// TIA Portal project "Pierwszy_projekt" (V16)

(* hardware
DEVICE "S71500/ET200MP station_1"  S7-1500 station
   slot 0: "Rail_0"  Rack  6ES7 590-1***0-0AA0
   slot 1: "PLC_1"  CPU 1518F-4 PN/DP  6ES7 518-4FP00-3AB0  V2.8
      slot 3: "CPU display_1"  6ES7591-1BA00-0AA0
      slot 32768: "PROFINET interface_1"  X1
         slot 32769: "Port_1"  X1 P1
         slot 32770: "Port_2"  X1 P2
      slot 33024: "PROFINET interface_2"  X2
         slot 33025: "Port_1"  X2 P1
      slot 33280: "PROFINET interface GBIT_3"  X3
         slot 33281: "Port_1"  X3 P1
      slot 33536: "DP interface_1"  X4
      slot 34817: "Virtual CP interface port_1"  Virtual CP interface port  Virtual CP interface port
*)

// ===== PLC "PLC_1"  CPU 1518F-4 PN/DP =====

VAR_GLOBAL   // PLC tag table "Default tag table"
   "System_Byte" AT %MB1 : Byte;
   "FirstScan" AT %M1.0 : Bool;
   "DiagStatusUpdate" AT %M1.1 : Bool;
   "AlwaysTRUE" AT %M1.2 : Bool;
   "AlwaysFALSE" AT %M1.3 : Bool;
   "System_Byte(1)" AT %MB1 : Byte;
   "Clock_Byte" AT %MB0 : Byte;
   "Clock_10Hz" AT %M0.0 : Bool;
   "Clock_5Hz" AT %M0.1 : Bool;
   "Clock_2.5Hz" AT %M0.2 : Bool;
   "Clock_2Hz" AT %M0.3 : Bool;
   "Clock_1.25Hz" AT %M0.4 : Bool;
   "Clock_1Hz" AT %M0.5 : Bool;
   "Clock_0.625Hz" AT %M0.6 : Bool;
   "Clock_0.5Hz" AT %M0.7 : Bool;
   "11-PLC01-MANUAL" AT %Q1.6 : Bool;
   "11-PLC01-AUTOMAT" AT %Q1.7 : Bool;
   "11-PLC01-DISPLAY01" AT %QD58 : Real;
   "Tag_1" AT %M3.0 : Bool;
   "Tag_2" AT %M2.0 : Bool;
   "Tag_3" AT %M2.1 : Bool;
   "Tag_4" AT %M2.2 : Bool;
   "Tag_5" AT %M2.3 : Bool;
   "Tag_6" AT %QD43 : Real;
   "Tag_7" AT %QD44 : Real;
   "Tag_8" AT %M2.5 : Bool;
   "Tag_9" AT %M2.6 : Bool;
   "Tag_10" AT %M2.7 : Bool;
   "Tag_11" AT %M250.4 : Bool;
   "Tag_12" AT %M650.0 : Bool;
   "Tag_13" AT %M654.0 : Bool;
   "Tag_14" AT %M2.4 : Bool;
   "Tag_15" AT %M3.5 : Bool;
END_VAR

VAR_GLOBAL   // PLC tag table "Tag table from XML_1"
   "11-PLC01-CNR01-SQ01" AT %I0.0 : Bool;
   "11-PLC01-CNR01-SQ02" AT %I0.1 : Bool;
   "11-PLC01-CNR01-ENC-A" AT %I0.2 : Bool;
   "11-PLC01-CNR01-ENC-B" AT %I0.3 : Bool;
   "11-PLC01-CNR02-SQ01" AT %I0.4 : Bool;
   "11-PLC01-CNR02-SQ02" AT %I0.5 : Bool;
   "11-PLC01-CNR02-ENC-A" AT %I0.6 : Bool;
   "11-PLC01-CNR02-ENC-B" AT %I0.7 : Bool;
   "11-PLC01-CNR03-SQ01" AT %I1.0 : Bool;
   "11-PLC01-CNR03-SQ02" AT %I1.1 : Bool;
   "11-PLC01-CNR03-ENC-A" AT %I1.2 : Bool;
   "11-PLC01-CNR03-ENC-B" AT %I1.3 : Bool;
   "11-PLC01-B01(START)" AT %I3.5 : Bool;
   "11-PLC01-B02(STOP)" AT %I3.6 : Bool;
   "11-PLC01-B03(RESET)" AT %I3.7 : Bool;
   "11-PLC01-B04(MANUAL)" AT %I4.0 : Bool;
   "11-PLC01-B05(AUTOMAT)" AT %I4.1 : Bool;
   "FACTORY I/O (Running)" AT %I4.2 : Bool;
   "FACTORY I/O (Paused)" AT %I4.3 : Bool;
   "FACTORY I/O (Reset)" AT %Q1.5 : Bool;
   "11-PLC01-PX01(START)" AT %Q0.0 : Bool;
   "11-PLC01-PX02(STOP)" AT %Q0.1 : Bool;
   "11-PLC01-PX03(RESET)" AT %Q0.2 : Bool;
   "11-PLC01-CNR01-EM01" AT %Q0.3 : Bool;
   "11-PLC01-CNR03-RE01" AT %Q0.4 : Bool;
   "FACTORY I/O (Run)" AT %Q1.3 : Bool;
   "FACTORY I/O (Pause)" AT %Q1.4 : Bool;
   "FACTORY I/O (Time Scale)" AT %ID34 : Real;
   "11-PLC01-CNR01" AT %QD30 : Real;
   "11-PLC01-CNR02" AT %QD34 : Real;
   "11-PLC01-CNR03" AT %QD38 : Real;
   "FACTORY I/O (Camera Position)" AT %QD54 : DInt;
END_VAR

VAR_GLOBAL   // PLC tag table "Tag table from XML_2"
   "11-PLC01-TT01-SQ01" AT %I1.4 : Bool;
   "11-PLC01-TT01-SQ02" AT %I1.5 : Bool;
   "11-PLC01-TT01-SQ03" AT %I1.6 : Bool;
   "11-PLC01-TT01-SQ04" AT %I1.7 : Bool;
   "11-PLC01-TT01-SQ05" AT %I2.0 : Bool;
   "11-PLC01-CNR04-SQ01" AT %I2.1 : Bool;
   "11-PLC01-CNR04-SQ02" AT %I2.2 : Bool;
   "11-PLC01-CNR04-ENC-A" AT %I2.3 : Bool;
   "11-PLC01-CNR04-ENC-B" AT %I2.4 : Bool;
   "11-PLC01-CNR05-SQ01" AT %I2.5 : Bool;
   "11-PLC01-CNR05-SQ02" AT %I2.6 : Bool;
   "11-PLC01-CNR05-ENC-A" AT %I2.7 : Bool;
   "11-PLC01-CNR05-ENC-B" AT %I3.0 : Bool;
   "11-PLC01-CNR06-SQ01" AT %I3.1 : Bool;
   "11-PLC01-CNR06-SQ02" AT %I3.2 : Bool;
   "11-PLC01-CNR06-ENC-A" AT %I3.3 : Bool;
   "11-PLC01-CNR06-ENC-B" AT %I3.4 : Bool;
   "11-PLC01-CNR04-RE01" AT %Q0.5 : Bool;
   "11-PLC01-CNR05-RE01" AT %Q0.6 : Bool;
   "11-PLC01-CNR06-RE01" AT %Q0.7 : Bool;
   "11-PLC01-TT01-LEFT" AT %Q2.0 : Bool;
   "11-PLC01-TT01-RIGHT" AT %Q2.1 : Bool;
   "11-PLC01-TT01-FORWARD" AT %Q2.2 : Bool;
   "11-PLC01-TT01-BACKWARD" AT %Q2.3 : Bool;
   "11-PLC01-CNR03-FLC01" AT %ID30 : Real;
   "11-PLC01-CNR04" AT %QD42 : Real;
   "11-PLC01-CNR05" AT %QD46 : Real;
   "11-PLC01-CNR06" AT %QD50 : Real;
END_VAR

DATA_BLOCK "Main_Safety_RTG1_DB"   // DB1, F_DB
{ S7_Optimized_Access := 'TRUE' }
NAME : FUSI
VERSION : 0.1
// stored: InstanceOfName Main_Safety_RTG1
"Main_Safety_RTG1"
BEGIN
END_DATA_BLOCK

DATA_BLOCK "FB_Conveyor_DB"   // DB2
{ S7_Optimized_Access := 'TRUE' }
VERSION : 0.1
// stored: InstanceOfName FB_Conveyor
"FB_Conveyor"
BEGIN
END_DATA_BLOCK

DATA_BLOCK "FB_Conveyor_DB_2"   // DB3
{ S7_Optimized_Access := 'TRUE' }
VERSION : 0.1
// stored: InstanceOfName FB_Conveyor
"FB_Conveyor"
BEGIN
END_DATA_BLOCK

DATA_BLOCK "DB_Manual"   // DB6
{ S7_Optimized_Access := 'TRUE' }
VERSION : 0.1
   VAR
      "11-CNR01-CONV" : Struct
         SelectManualMode : Bool := TRUE;
         StartStop : Bool := TRUE;
         SetSpeed : Int := 80;
      END_STRUCT;
      "11-CNR02-CONV" : Struct
         SelectManual : Bool := TRUE;
         StartStop : Bool := TRUE;
         SetSpeed : Int := 80;
      END_STRUCT;
      "11-CNRO3-CONV" : Struct
         SelectManualMode : Bool := TRUE;
         StartStop : Bool := TRUE;
         SetSpeed : Int := 100;
      END_STRUCT;
   END_VAR
BEGIN
END_DATA_BLOCK

DATA_BLOCK "FB_Inverter_DB"   // DB7
{ S7_Optimized_Access := 'TRUE' }
VERSION : 0.1
// stored: InstanceOfName FB_Inverter
"FB_Inverter"
BEGIN
END_DATA_BLOCK

DATA_BLOCK "FB_Conveyor_DB_1"   // DB8
{ S7_Optimized_Access := 'TRUE' }
VERSION : 0.1
// stored: InstanceOfName FB_Conveyor
"FB_Conveyor"
BEGIN
END_DATA_BLOCK

DATA_BLOCK "DB_Signals"   // DB9
{ S7_Optimized_Access := 'TRUE' }
VERSION : 0.1
   VAR
      "11-CNR01-VFD" : Struct
         RunForward : Bool;
         RunRevers : Bool;
         ConveyorSpeedSetPoint : Real;
      END_STRUCT;
      "11-CNR02-VFD" : Struct
         RunForward : Bool;
         RunRevers : Bool;
         ConveyorSpeedSetPoint : Real;
      END_STRUCT;
      "11-CNR03-VFD" : Struct
         RunForward : Bool;
         RunRevrs : Bool;
         ConveyorSpeedSetPoint : Real;
      END_STRUCT;
   END_VAR
BEGIN
END_DATA_BLOCK

DATA_BLOCK "DB_Configuration"   // DB10
{ S7_Optimized_Access := 'TRUE' }
VERSION : 0.1
   VAR
      "11-CNR01-VFD" : Struct
         InterlockForwad : Bool := TRUE;
         InterockReverse : Bool;
      END_STRUCT;
      "11-CNR02-VDF" : Struct
         InterlockForwad : Bool := TRUE;
         InterockReverse : Bool;
      END_STRUCT;
      "11-CNR03-VDF" : Struct
         InterlockForwad : Bool := TRUE;
         InterockReverse : Bool;
      END_STRUCT;
   END_VAR
BEGIN
END_DATA_BLOCK

DATA_BLOCK "FB_Inverter_DB_1"   // DB11
{ S7_Optimized_Access := 'TRUE' }
VERSION : 0.1
// stored: InstanceOfName FB_Inverter
"FB_Inverter"
BEGIN
END_DATA_BLOCK

DATA_BLOCK "FB_Inverter_DB_2"   // DB12
{ S7_Optimized_Access := 'TRUE' }
VERSION : 0.1
// stored: InstanceOfName FB_Inverter
"FB_Inverter"
BEGIN
END_DATA_BLOCK

DATA_BLOCK "FB_TurnTable_DB"   // DB13
{ S7_Optimized_Access := 'TRUE' }
VERSION : 0.1
// stored: InstanceOfName FB_TurnTable
"FB_TurnTable"
BEGIN
END_DATA_BLOCK

DATA_BLOCK "FB_Control_DB"   // DB14
{ S7_Optimized_Access := 'TRUE' }
VERSION : 0.1
// stored: InstanceOfName FB_Control
"FB_Control"
BEGIN
END_DATA_BLOCK

DATA_BLOCK "FB_Control_DB_1"   // DB15
{ S7_Optimized_Access := 'TRUE' }
VERSION : 0.1
// stored: InstanceOfName FB_Control
"FB_Control"
BEGIN
END_DATA_BLOCK

DATA_BLOCK "DB_Control"   // DB16
{ S7_Optimized_Access := 'TRUE' }
VERSION : 0.1
   VAR
      StartCommand : Bool := false;
      StopCommand : Bool;
      StartFeedback : Bool := false;
      StopFeedback : Bool;
      ManualFeedback : Bool;
   END_VAR
BEGIN
END_DATA_BLOCK

DATA_BLOCK "IDB_FIFO"   // DB20
{ S7_Optimized_Access := 'TRUE' }
VERSION : 0.1
   VAR
      Static_1 : Array[0..10] of Real;
      Arrey_return : Int;
      Array_Dest : Array[0..10] of Real;
      Array_Input : Array[0..5] of Real;
      Array_endofqueue : Array[0..10] of Real;
   END_VAR
BEGIN
END_DATA_BLOCK

DATA_BLOCK "FD_FIFO_DB"   // DB22
{ S7_Optimized_Access := 'TRUE' }
VERSION : 0.1
// stored: InstanceOfName FD_FIFO
"FD_FIFO"
BEGIN
END_DATA_BLOCK

DATA_BLOCK "FB_Chute_DB- smallpackage"   // DB25
{ S7_Optimized_Access := 'TRUE' }
VERSION : 0.1
// stored: InstanceOfName FB_Chute
"FB_Chute"
BEGIN
END_DATA_BLOCK

DATA_BLOCK "FB_Chute_DB-mediumpackage"   // DB26
{ S7_Optimized_Access := 'TRUE' }
VERSION : 0.1
// stored: InstanceOfName FB_Chute
"FB_Chute"
BEGIN
END_DATA_BLOCK

DATA_BLOCK "FB_Chute_DB-bigpackage"   // DB27
{ S7_Optimized_Access := 'TRUE' }
VERSION : 0.1
// stored: InstanceOfName FB_Chute
"FB_Chute"
BEGIN
END_DATA_BLOCK

DATA_BLOCK "DB_Chute"   // DB30
{ S7_Optimized_Access := 'TRUE' }
VERSION : 0.1
   VAR
      "Small Package" : Int;
      "Medium Package" : Int;
      "Big Package" : Int;
   END_VAR
BEGIN
END_DATA_BLOCK

// folder: System blocks/Program resources

DATA_BLOCK "StartButtonCount_DB"   // DB4
{ S7_Optimized_Access := 'TRUE' }
AUTHOR : Simatic
FAMILY : IEC
NAME : CNTR
VERSION : 1.0
// stored: InstanceOfName IEC_COUNTER
"IEC_COUNTER"
BEGIN
END_DATA_BLOCK

DATA_BLOCK "DelayStartDB"   // DB5
{ S7_Optimized_Access := 'TRUE' }
AUTHOR : Simatic
FAMILY : IEC
NAME : IEC_TMR
VERSION : 1.0
// stored: InstanceOfName IEC_TIMER
"IEC_TIMER"
BEGIN
END_DATA_BLOCK

DATA_BLOCK "IEC_Counter_0_DB"   // DB17
{ S7_Optimized_Access := 'TRUE' }
AUTHOR : Simatic
FAMILY : IEC
NAME : CNTR
VERSION : 1.0
// stored: InstanceOfName IEC_COUNTER
"IEC_COUNTER"
BEGIN
END_DATA_BLOCK

DATA_BLOCK "IEC_Counter_0_DB_1"   // DB18
{ S7_Optimized_Access := 'TRUE' }
AUTHOR : Simatic
FAMILY : IEC
NAME : CNTR
VERSION : 1.0
// stored: InstanceOfName IEC_COUNTER
"IEC_COUNTER"
BEGIN
END_DATA_BLOCK

DATA_BLOCK "IEC_Counter_0_DB_2"   // DB19
{ S7_Optimized_Access := 'TRUE' }
AUTHOR : Simatic
FAMILY : IEC
NAME : CNTR
VERSION : 1.0
// stored: InstanceOfName IEC_COUNTER
"IEC_COUNTER"
BEGIN
END_DATA_BLOCK

DATA_BLOCK "IEC_Counter_0_DB_3"   // DB21
{ S7_Optimized_Access := 'TRUE' }
AUTHOR : Simatic
FAMILY : IEC
NAME : CNTR
VERSION : 1.0
// stored: InstanceOfName IEC_COUNTER
"IEC_COUNTER"
BEGIN
END_DATA_BLOCK

DATA_BLOCK "IEC_Counter_0_DB_4"   // DB24
{ S7_Optimized_Access := 'TRUE' }
AUTHOR : Simatic
FAMILY : IEC
NAME : CNTR
VERSION : 1.0
// stored: InstanceOfName IEC_COUNTER
"IEC_COUNTER"
BEGIN
END_DATA_BLOCK

DATA_BLOCK "IEC_Counter_0_DB_5"   // DB28
{ S7_Optimized_Access := 'TRUE' }
AUTHOR : Simatic
FAMILY : IEC
NAME : CNTR
VERSION : 1.0
// stored: InstanceOfName IEC_COUNTER
"IEC_COUNTER"
BEGIN
END_DATA_BLOCK

DATA_BLOCK "IEC_Counter_0_DB_6"   // DB29
{ S7_Optimized_Access := 'TRUE' }
AUTHOR : Simatic
FAMILY : IEC
NAME : CNTR
VERSION : 1.0
// stored: InstanceOfName IEC_COUNTER
"IEC_COUNTER"
BEGIN
END_DATA_BLOCK

// folder: (top level)

FUNCTION_BLOCK "Main_Safety_RTG1"   // FB1, F_FBD
{ S7_Optimized_Access := 'TRUE' }
BEGIN
END_FUNCTION_BLOCK

FUNCTION_BLOCK "FB_Conveyor"   // FB2, LAD
{ S7_Optimized_Access := 'TRUE' }
VERSION : 0.1
   VAR_INPUT
      ir_ConveyorSpeed : Real;
      ix_PEC_BOS : Bool;
      ix_PEC_EOS : Bool;
   END_VAR
   VAR_OUTPUT
      qx_FlowStop : Bool;
   END_VAR
   VAR_IN_OUT
      iqx_StartStop : Bool;
      iqi_SetSpeed : Int;
      iqx_SelectManualMode : Bool;
      iqr_InverterSpeedSetpoint : Real;
      iqx_InverterRunForward : Bool;
      iqx_InverterRunReverse : Bool;
      iqx_ControlStart : Bool;
      iqx_ControlStop : Bool;
      iqx_ControlManual : Bool;
   END_VAR
   VAR
      sx_manual : Bool;
      sx_Automatic : Bool;
      sx_FlowStop : Bool;
   END_VAR
   VAR_TEMP
      tr_SpeedPoint : Real;
      tr_SpeedProcent : Int;
   END_VAR
   VAR_TEMP   // added for the SCL form of the ladder/FBD networks
      _w1 : Bool;
      _w2 : Bool;
      _w3 : Bool;
   END_VAR
BEGIN

REGION Network 1
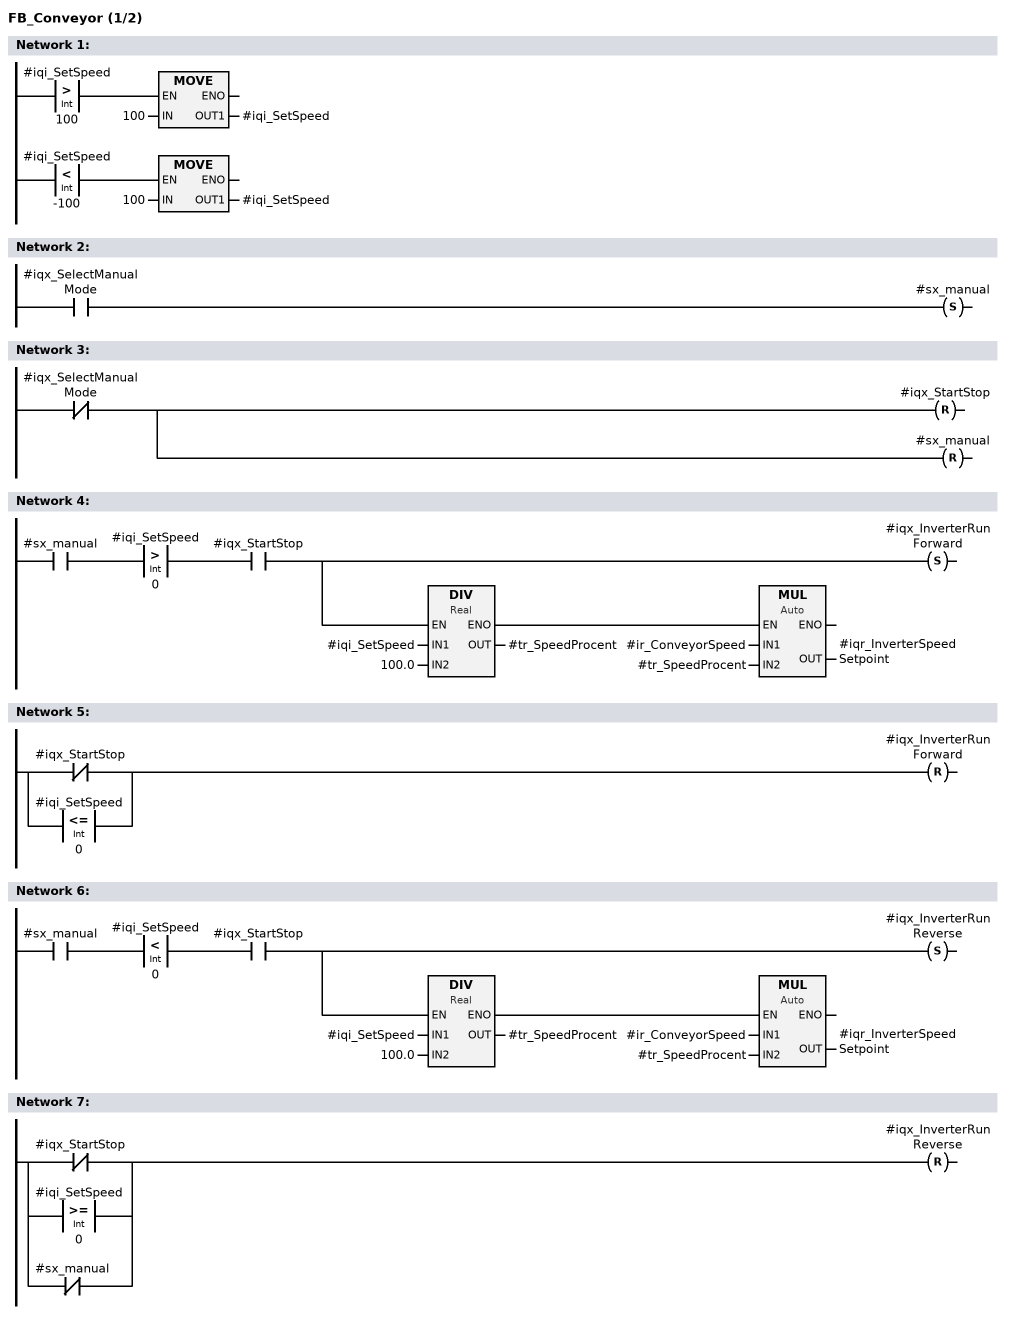
   RUNG wire#powerrail
      { S7_Templates := "SrcType := Int" } GT_Contact(in1 := #iqi_SetSpeed, in2 := 100)
      Move(in := 100, out1 => #iqi_SetSpeed)
   END_RUNG
   RUNG wire#powerrail
      { S7_Templates := "SrcType := Int" } LT_Contact(in1 := #iqi_SetSpeed, in2 := -100)
      Move(in := 100, out1 => #iqi_SetSpeed)
   END_RUNG
   // the same network as SCL:
   IF #iqi_SetSpeed > 100 THEN #iqi_SetSpeed := 100; END_IF;
   IF #iqi_SetSpeed < (-100) THEN #iqi_SetSpeed := 100; END_IF;
END_REGION

REGION Network 2
   RUNG wire#powerrail
      Contact( #iqx_SelectManualMode )
      S_Coil( #sx_manual )
   END_RUNG
   // the same network as SCL:
   IF #iqx_SelectManualMode THEN #sx_manual := TRUE; END_IF;
END_REGION

REGION Network 3
   RUNG wire#powerrail
      I_Contact( #iqx_SelectManualMode )
      wire#w1
      R_Coil( #iqx_StartStop )
   END_RUNG
   RUNG wire#w1
      R_Coil( #sx_manual )
   END_RUNG
   // the same network as SCL:
   IF NOT #iqx_SelectManualMode THEN
       #iqx_StartStop := FALSE;
       #sx_manual := FALSE;
   END_IF;
END_REGION

REGION Network 4
   RUNG wire#powerrail
      Contact( #sx_manual )
      { S7_Templates := "SrcType := Int" } GT_Contact(in1 := #iqi_SetSpeed, in2 := 0)
      Contact( #iqx_StartStop )
      wire#w1
      S_Coil( #iqx_InverterRunForward )
   END_RUNG
   RUNG wire#w1
      { S7_Templates := "SrcType := Real" } Div(in1 := #iqi_SetSpeed, in2 := 100.0, out => #tr_SpeedProcent)
      Mul(in1 := #ir_ConveyorSpeed, in2 := #tr_SpeedProcent, out => #iqr_InverterSpeedSetpoint)
   END_RUNG
   // the same network as SCL:
   IF #sx_manual AND (#iqi_SetSpeed > 0) AND #iqx_StartStop THEN
       #iqx_InverterRunForward := TRUE;
       #tr_SpeedProcent := #iqi_SetSpeed / 100.0;
       #iqr_InverterSpeedSetpoint := #ir_ConveyorSpeed * #tr_SpeedProcent;
   END_IF;
END_REGION

REGION Network 5
   RUNG wire#powerrail
      I_Contact( #iqx_StartStop )
      wire#w1
      R_Coil( #iqx_InverterRunForward )
   END_RUNG
   RUNG wire#powerrail
      { S7_Templates := "SrcType := Int" } LE_Contact(in1 := #iqi_SetSpeed, in2 := 0)
   END_RUNG wire#w1
   // the same network as SCL:
   IF NOT #iqx_StartStop OR (#iqi_SetSpeed <= 0) THEN #iqx_InverterRunForward := FALSE; END_IF;
END_REGION

REGION Network 6
   RUNG wire#powerrail
      Contact( #sx_manual )
      { S7_Templates := "SrcType := Int" } LT_Contact(in1 := #iqi_SetSpeed, in2 := 0)
      Contact( #iqx_StartStop )
      wire#w1
      S_Coil( #iqx_InverterRunReverse )
   END_RUNG
   RUNG wire#w1
      { S7_Templates := "SrcType := Real" } Div(in1 := #iqi_SetSpeed, in2 := 100.0, out => #tr_SpeedProcent)
      Mul(in1 := #ir_ConveyorSpeed, in2 := #tr_SpeedProcent, out => #iqr_InverterSpeedSetpoint)
   END_RUNG
   // the same network as SCL:
   IF #sx_manual AND (#iqi_SetSpeed < 0) AND #iqx_StartStop THEN
       #iqx_InverterRunReverse := TRUE;
       #tr_SpeedProcent := #iqi_SetSpeed / 100.0;
       #iqr_InverterSpeedSetpoint := #ir_ConveyorSpeed * #tr_SpeedProcent;
   END_IF;
END_REGION

REGION Network 7
   RUNG wire#powerrail
      I_Contact( #iqx_StartStop )
      wire#w1
      R_Coil( #iqx_InverterRunReverse )
   END_RUNG
   RUNG wire#powerrail
      { S7_Templates := "SrcType := Int" } GE_Contact(in1 := #iqi_SetSpeed, in2 := 0)
   END_RUNG wire#w1
   RUNG wire#powerrail
      I_Contact( #sx_manual )
   END_RUNG wire#w1
   // the same network as SCL:
   IF NOT #iqx_StartStop OR (#iqi_SetSpeed >= 0) OR NOT #sx_manual THEN
       #iqx_InverterRunReverse := FALSE;
   END_IF;
END_REGION

REGION Network 8
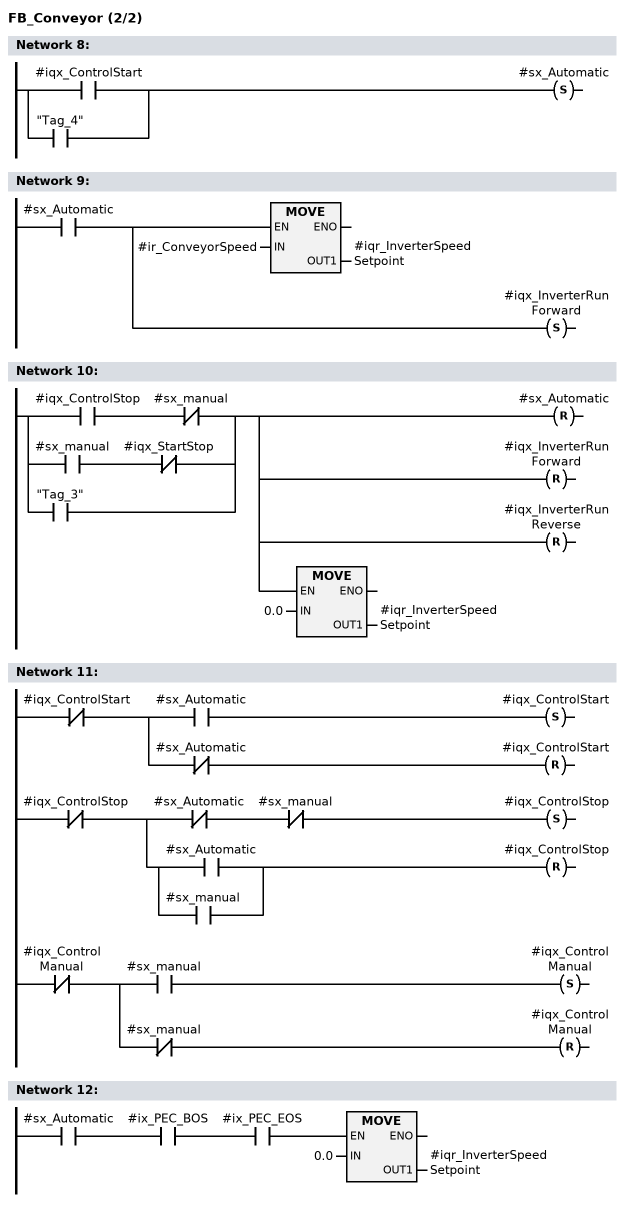
   RUNG wire#powerrail
      Contact( #iqx_ControlStart )
      wire#w1
      S_Coil( #sx_Automatic )
   END_RUNG
   RUNG wire#powerrail
      Contact( "Tag_4" )
   END_RUNG wire#w1
   // the same network as SCL:
   IF #iqx_ControlStart OR "Tag_4" THEN #sx_Automatic := TRUE; END_IF;
END_REGION

REGION Network 9
   RUNG wire#powerrail
      Contact( #sx_Automatic )
      wire#w1
      Move(in := #ir_ConveyorSpeed, out1 => #iqr_InverterSpeedSetpoint)
   END_RUNG
   RUNG wire#w1
      S_Coil( #iqx_InverterRunForward )
   END_RUNG
   // the same network as SCL:
   IF #sx_Automatic THEN
       #iqr_InverterSpeedSetpoint := #ir_ConveyorSpeed;
       #iqx_InverterRunForward := TRUE;
   END_IF;
END_REGION

REGION Network 10
   RUNG wire#powerrail
      Contact( #iqx_ControlStop )
      I_Contact( #sx_manual )
      wire#w1
      R_Coil( #sx_Automatic )
   END_RUNG
   RUNG wire#powerrail
      Contact( #sx_manual )
      I_Contact( #iqx_StartStop )
   END_RUNG wire#w1
   RUNG wire#powerrail
      Contact( "Tag_3" )
   END_RUNG wire#w1
   RUNG wire#w1
      R_Coil( #iqx_InverterRunForward )
   END_RUNG
   RUNG wire#w1
      R_Coil( #iqx_InverterRunReverse )
   END_RUNG
   RUNG wire#w1
      Move(in := 0.0, out1 => #iqr_InverterSpeedSetpoint)
   END_RUNG
   // the same network as SCL:
   IF (#iqx_ControlStop AND NOT #sx_manual) OR (#sx_manual AND NOT #iqx_StartStop) OR "Tag_3" THEN
       #sx_Automatic := FALSE;
       #iqx_InverterRunForward := FALSE;
       #iqx_InverterRunReverse := FALSE;
       #iqr_InverterSpeedSetpoint := 0.0;
   END_IF;
END_REGION

REGION Network 11
   RUNG wire#powerrail
      I_Contact( #iqx_ControlStart )
      wire#w1
      Contact( #sx_Automatic )
      S_Coil( #iqx_ControlStart )
   END_RUNG
   RUNG wire#w1
      I_Contact( #sx_Automatic )
      R_Coil( #iqx_ControlStart )
   END_RUNG
   RUNG wire#powerrail
      I_Contact( #iqx_ControlStop )
      wire#w2
      I_Contact( #sx_Automatic )
      I_Contact( #sx_manual )
      S_Coil( #iqx_ControlStop )
   END_RUNG
   RUNG wire#w2
      Contact( #sx_Automatic )
      wire#w3
      R_Coil( #iqx_ControlStop )
   END_RUNG
   RUNG wire#w2
      Contact( #sx_manual )
   END_RUNG wire#w3
   RUNG wire#powerrail
      I_Contact( #iqx_ControlManual )
      wire#w4
      Contact( #sx_manual )
      S_Coil( #iqx_ControlManual )
   END_RUNG
   RUNG wire#w4
      I_Contact( #sx_manual )
      R_Coil( #iqx_ControlManual )
   END_RUNG
   // the same network as SCL:
   #_w1 := NOT #iqx_ControlStart;
   IF NOT #iqx_ControlStart AND #sx_Automatic THEN #iqx_ControlStart := TRUE; END_IF;
   IF #_w1 AND NOT #sx_Automatic THEN #iqx_ControlStart := FALSE; END_IF;
   #_w2 := NOT #iqx_ControlStop;
   IF NOT #iqx_ControlStop AND NOT #sx_Automatic AND NOT #sx_manual THEN #iqx_ControlStop := TRUE; END_IF;
   IF #_w2 AND (#sx_Automatic OR #sx_manual) THEN #iqx_ControlStop := FALSE; END_IF;
   #_w3 := NOT #iqx_ControlManual;
   IF NOT #iqx_ControlManual AND #sx_manual THEN #iqx_ControlManual := TRUE; END_IF;
   IF #_w3 AND NOT #sx_manual THEN #iqx_ControlManual := FALSE; END_IF;
END_REGION

REGION Network 12
   RUNG wire#powerrail
      Contact( #sx_Automatic )
      Contact( #ix_PEC_BOS )
      Contact( #ix_PEC_EOS )
      Move(in := 0.0, out1 => #iqr_InverterSpeedSetpoint)
   END_RUNG
   // the same network as SCL:
   IF #sx_Automatic AND #ix_PEC_BOS AND #ix_PEC_EOS THEN #iqr_InverterSpeedSetpoint := 0.0; END_IF;
END_REGION
END_FUNCTION_BLOCK

FUNCTION_BLOCK "FB_Inverter"   // FB3, LAD
{ S7_Optimized_Access := 'TRUE' }
VERSION : 0.1
   VAR_INPUT
      ix_InterlockForward : Bool;
      Ix_InterlockReverse : Bool;
      Ir_ConveyorSpeedSetpoint : Real;
   END_VAR
   VAR_OUTPUT
      qr_InverterSpeed : Real;
   END_VAR
   VAR_IN_OUT
      iqx_InverterRunForward : Bool;
      iqx_InverterRunReverse : Bool;
   END_VAR
   VAR
      sx_RunForward : Bool;
      sx_RunReverse : Bool;
   END_VAR
BEGIN

REGION Network 1
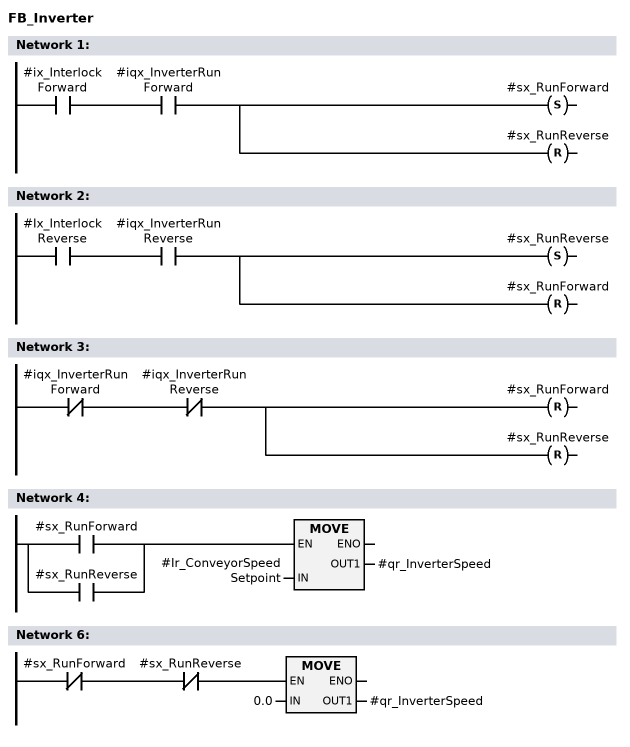
   RUNG wire#powerrail
      Contact( #ix_InterlockForward )
      Contact( #iqx_InverterRunForward )
      wire#w1
      S_Coil( #sx_RunForward )
   END_RUNG
   RUNG wire#w1
      R_Coil( #sx_RunReverse )
   END_RUNG
   // the same network as SCL:
   IF #ix_InterlockForward AND #iqx_InverterRunForward THEN
       #sx_RunForward := TRUE;
       #sx_RunReverse := FALSE;
   END_IF;
END_REGION

REGION Network 2
   RUNG wire#powerrail
      Contact( #Ix_InterlockReverse )
      Contact( #iqx_InverterRunReverse )
      wire#w1
      S_Coil( #sx_RunReverse )
   END_RUNG
   RUNG wire#w1
      R_Coil( #sx_RunForward )
   END_RUNG
   // the same network as SCL:
   IF #Ix_InterlockReverse AND #iqx_InverterRunReverse THEN
       #sx_RunReverse := TRUE;
       #sx_RunForward := FALSE;
   END_IF;
END_REGION

REGION Network 3
   RUNG wire#powerrail
      I_Contact( #iqx_InverterRunForward )
      I_Contact( #iqx_InverterRunReverse )
      wire#w1
      R_Coil( #sx_RunForward )
   END_RUNG
   RUNG wire#w1
      R_Coil( #sx_RunReverse )
   END_RUNG
   // the same network as SCL:
   IF NOT #iqx_InverterRunForward AND NOT #iqx_InverterRunReverse THEN
       #sx_RunForward := FALSE;
       #sx_RunReverse := FALSE;
   END_IF;
END_REGION

REGION Network 4
   RUNG wire#powerrail
      Contact( #sx_RunForward )
      wire#w1
      Move(in := #Ir_ConveyorSpeedSetpoint, out1 => #qr_InverterSpeed)
   END_RUNG
   RUNG wire#powerrail
      Contact( #sx_RunReverse )
   END_RUNG wire#w1
   // the same network as SCL:
   IF #sx_RunForward OR #sx_RunReverse THEN #qr_InverterSpeed := #Ir_ConveyorSpeedSetpoint; END_IF;
END_REGION

REGION Network 6
   RUNG wire#powerrail
      I_Contact( #sx_RunForward )
      I_Contact( #sx_RunReverse )
      Move(in := 0.0, out1 => #qr_InverterSpeed)
   END_RUNG
   // the same network as SCL:
   IF NOT #sx_RunForward AND NOT #sx_RunReverse THEN #qr_InverterSpeed := 0.0; END_IF;
END_REGION
END_FUNCTION_BLOCK

FUNCTION_BLOCK "FB_Control"   // FB4, LAD
{ S7_Optimized_Access := 'TRUE' }
VERSION : 0.1
   VAR_IN_OUT
      iqx_StartHMICommand : Bool;
      iqx_StopHMICommand : Bool;
      iqx_StartFeedback : Bool;
      iqx_StopFeedback : Bool;
      iqx_ManualFeedback : Bool;
   END_VAR
   VAR
      sudi_SignalingTime : Time := T#300ms;
      sx_StartRequest : Bool;
      s_TON_Timer : TON_TIME;
   END_VAR
BEGIN

REGION Network 1
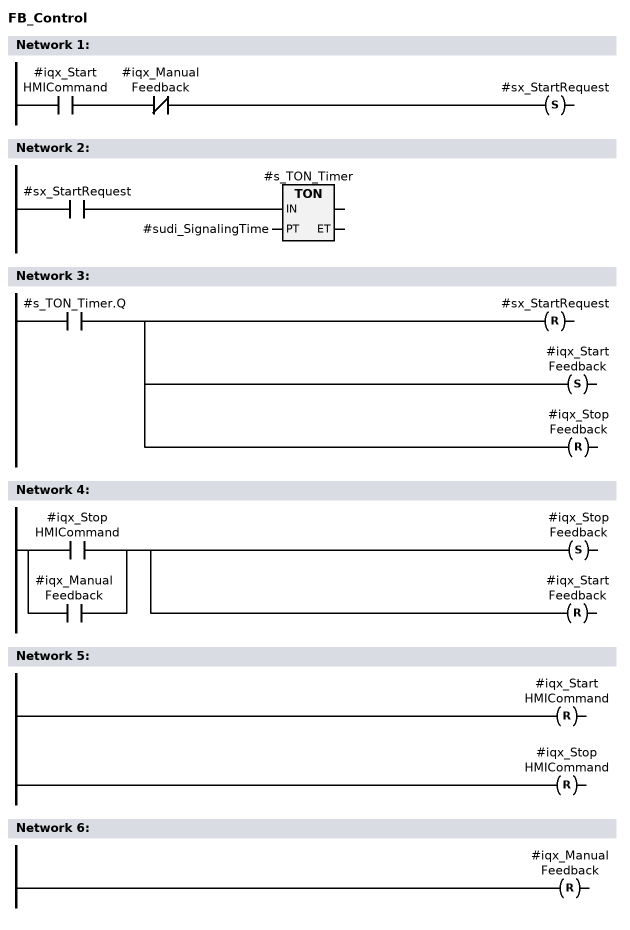
   RUNG wire#powerrail
      Contact( #iqx_StartHMICommand )
      I_Contact( #iqx_ManualFeedback )
      S_Coil( #sx_StartRequest )
   END_RUNG
   // the same network as SCL:
   IF #iqx_StartHMICommand AND NOT #iqx_ManualFeedback THEN #sx_StartRequest := TRUE; END_IF;
END_REGION

REGION Network 2
   #s_TON_Timer(IN := #sx_StartRequest, PT := #sudi_SignalingTime);   // TON
END_REGION

REGION Network 3
   RUNG wire#powerrail
      Contact( #s_TON_Timer.Q )
      wire#w1
      R_Coil( #sx_StartRequest )
   END_RUNG
   RUNG wire#w1
      S_Coil( #iqx_StartFeedback )
   END_RUNG
   RUNG wire#w1
      R_Coil( #iqx_StopFeedback )
   END_RUNG
   // the same network as SCL:
   IF #s_TON_Timer.Q THEN
       #sx_StartRequest := FALSE;
       #iqx_StartFeedback := TRUE;
       #iqx_StopFeedback := FALSE;
   END_IF;
END_REGION

REGION Network 4
   RUNG wire#powerrail
      Contact( #iqx_StopHMICommand )
      wire#w1
      S_Coil( #iqx_StopFeedback )
   END_RUNG
   RUNG wire#powerrail
      Contact( #iqx_ManualFeedback )
   END_RUNG wire#w1
   RUNG wire#w1
      R_Coil( #iqx_StartFeedback )
   END_RUNG
   // the same network as SCL:
   IF #iqx_StopHMICommand OR #iqx_ManualFeedback THEN
       #iqx_StopFeedback := TRUE;
       #iqx_StartFeedback := FALSE;
   END_IF;
END_REGION

REGION Network 5
   RUNG wire#powerrail
      R_Coil( #iqx_StartHMICommand )
   END_RUNG
   RUNG wire#powerrail
      R_Coil( #iqx_StopHMICommand )
   END_RUNG
   // the same network as SCL:
   #iqx_StartHMICommand := FALSE;
   #iqx_StopHMICommand := FALSE;
END_REGION

REGION Network 6
   RUNG wire#powerrail
      R_Coil( #iqx_ManualFeedback )
   END_RUNG
   // the same network as SCL:
   #iqx_ManualFeedback := FALSE;
END_REGION
END_FUNCTION_BLOCK

FUNCTION_BLOCK "FB_TurnTable"   // FB5, LAD
{ S7_Optimized_Access := 'TRUE' }
VERSION : 0.1
   VAR_INPUT
      ix_PEC_BigPackage_1 : Bool;
      ix_PEC_BigPackage_2 : Bool;
      ix_PEC_MediumPackage_1 : Bool;
      ix_PEC_MediumPackage_2 : Bool;
      ix_PEC_SmallPackage_1 : Bool;
      ix_PEC_SmallPackage_2 : Bool;
      ix_PEC_DetectPackage_1 : Bool;
      ix_PEC_DetectPackage_2 : Bool;
      ix_PEC_90Degree : Bool;
      ix_PEC_DiagonallyTT : Bool;
      ix_Reset : Bool;
   END_VAR
   VAR_OUTPUT
      qx_TTForward : Bool;
      qx_TTBackward : Bool;
      qx_TTLeft : Bool;
      qx_TTRight : Bool;
   END_VAR
   VAR_IN_OUT
      sx_Automatic_2 : Bool;
   END_VAR
   VAR
      sx_Automatic : Bool;
   END_VAR
   VAR_TEMP   // added for the SCL form of the ladder/FBD networks
      _w1 : Bool;
   END_VAR
BEGIN

REGION Network 1
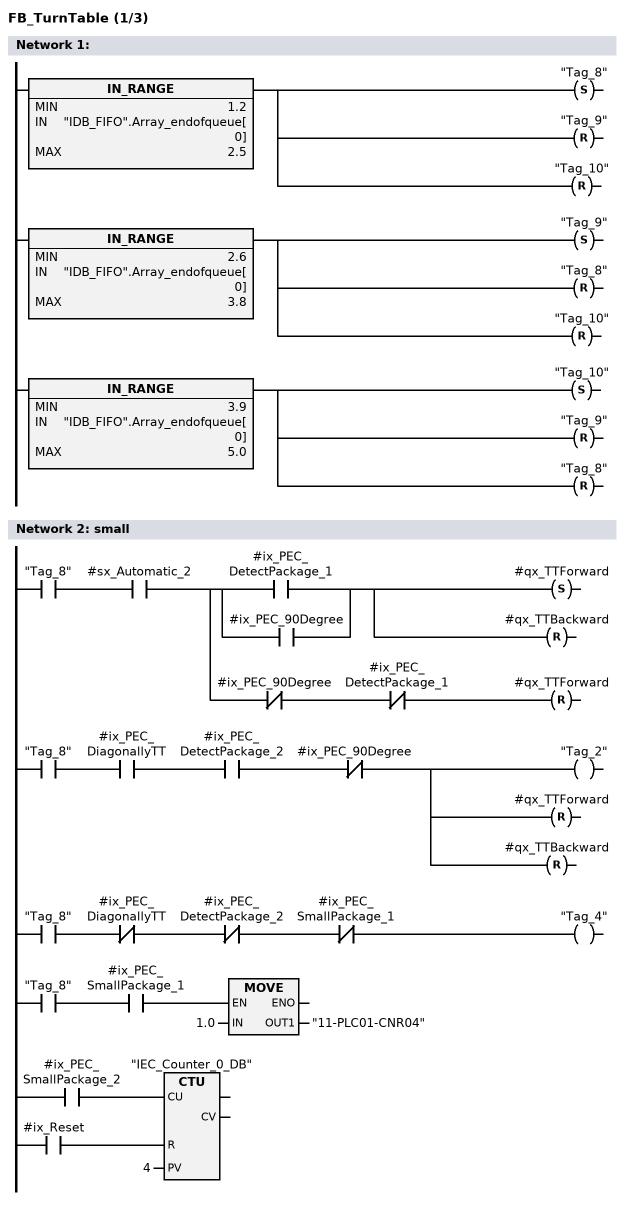
   RUNG wire#powerrail
      { S7_Templates := "SrcType := Real" } InRange(min := 1.2, in := "IDB_FIFO".Array_endofqueue[0], max := 2.5)
      wire#w1
      S_Coil( "Tag_8" )
   END_RUNG
   RUNG wire#w1
      R_Coil( "Tag_9" )
   END_RUNG
   RUNG wire#w1
      R_Coil( "Tag_10" )
   END_RUNG
   RUNG wire#powerrail
      { S7_Templates := "SrcType := Real" } InRange(min := 2.6, in := "IDB_FIFO".Array_endofqueue[0], max := 3.8)
      wire#w2
      S_Coil( "Tag_9" )
   END_RUNG
   RUNG wire#w2
      R_Coil( "Tag_8" )
   END_RUNG
   RUNG wire#w2
      R_Coil( "Tag_10" )
   END_RUNG
   RUNG wire#powerrail
      { S7_Templates := "SrcType := Real" } InRange(min := 3.9, in := "IDB_FIFO".Array_endofqueue[0], max := 5.0)
      wire#w3
      S_Coil( "Tag_10" )
   END_RUNG
   RUNG wire#w3
      R_Coil( "Tag_9" )
   END_RUNG
   RUNG wire#w3
      R_Coil( "Tag_8" )
   END_RUNG
   // the same network as SCL:
   IF (1.2 <= "IDB_FIFO".Array_endofqueue[0]) AND ("IDB_FIFO".Array_endofqueue[0] <= 2.5) THEN
       "Tag_8" := TRUE;
       "Tag_9" := FALSE;
       "Tag_10" := FALSE;
   END_IF;
   IF (2.6 <= "IDB_FIFO".Array_endofqueue[0]) AND ("IDB_FIFO".Array_endofqueue[0] <= 3.8) THEN
       "Tag_9" := TRUE;
       "Tag_8" := FALSE;
       "Tag_10" := FALSE;
   END_IF;
   IF (3.9 <= "IDB_FIFO".Array_endofqueue[0]) AND ("IDB_FIFO".Array_endofqueue[0] <= 5.0) THEN
       "Tag_10" := TRUE;
       "Tag_9" := FALSE;
       "Tag_8" := FALSE;
   END_IF;
END_REGION

REGION Network 2: small
   #_w1 := "Tag_8" AND #sx_Automatic_2;
   IF #_w1 AND (#ix_PEC_DetectPackage_1 OR #ix_PEC_90Degree) THEN
       #qx_TTForward := TRUE;
       #qx_TTBackward := FALSE;
   END_IF;
   IF #_w1 AND NOT #ix_PEC_90Degree AND NOT #ix_PEC_DetectPackage_1 THEN #qx_TTForward := FALSE; END_IF;
   "Tag_2" := "Tag_8" AND #ix_PEC_DiagonallyTT AND #ix_PEC_DetectPackage_2 AND NOT #ix_PEC_90Degree;
   IF "Tag_2" THEN
       #qx_TTForward := FALSE;
       #qx_TTBackward := FALSE;
   END_IF;
   "Tag_4" := "Tag_8" AND NOT #ix_PEC_DiagonallyTT AND NOT #ix_PEC_DetectPackage_2 AND NOT #ix_PEC_SmallPackage_1;
   IF "Tag_8" AND #ix_PEC_SmallPackage_1 THEN "11-PLC01-CNR04" := 1.0; END_IF;
   "IEC_Counter_0_DB".CTU(CU := #ix_PEC_SmallPackage_2, R := #ix_Reset, PV := 4);
END_REGION

REGION Network 3: medium
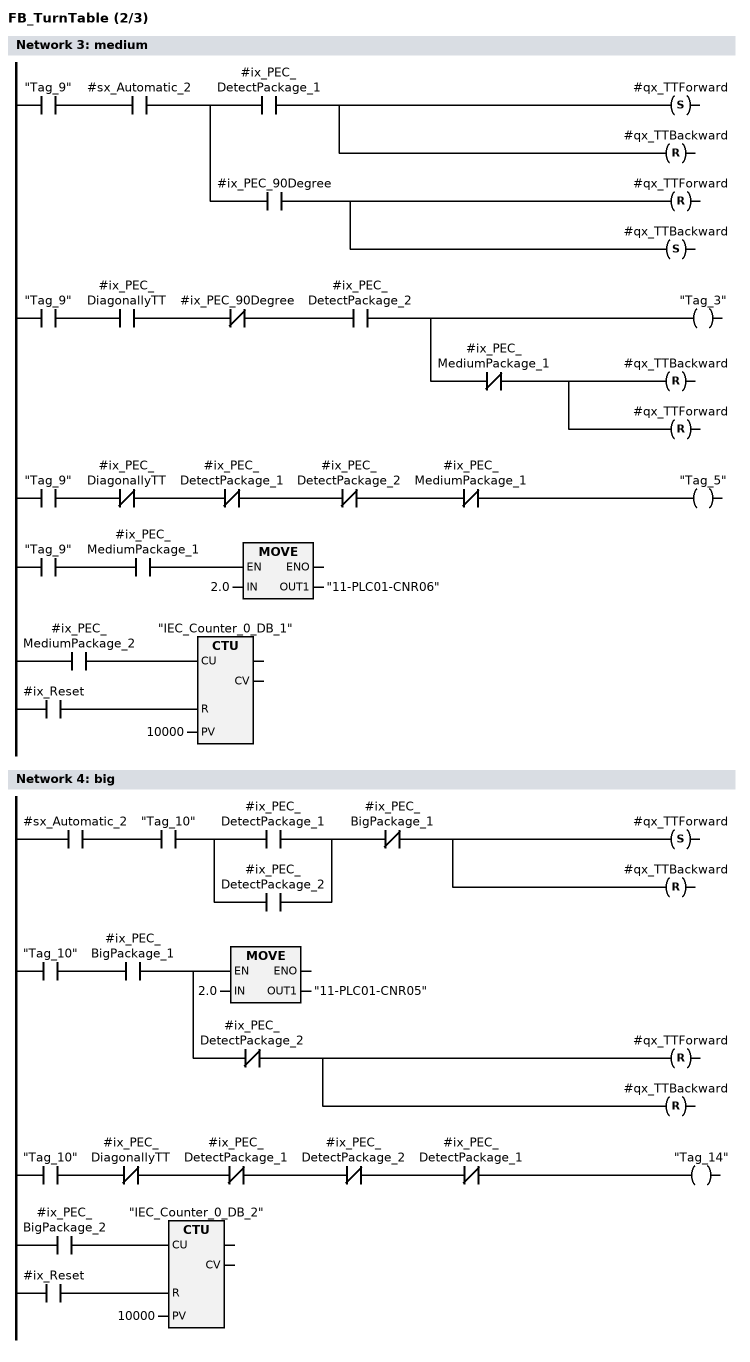
   #_w1 := "Tag_9" AND #sx_Automatic_2;
   IF #_w1 AND #ix_PEC_DetectPackage_1 THEN
       #qx_TTForward := TRUE;
       #qx_TTBackward := FALSE;
   END_IF;
   IF #_w1 AND #ix_PEC_90Degree THEN
       #qx_TTForward := FALSE;
       #qx_TTBackward := TRUE;
   END_IF;
   "Tag_3" := "Tag_9" AND #ix_PEC_DiagonallyTT AND NOT #ix_PEC_90Degree AND #ix_PEC_DetectPackage_2;
   IF "Tag_3" AND NOT #ix_PEC_MediumPackage_1 THEN
       #qx_TTBackward := FALSE;
       #qx_TTForward := FALSE;
   END_IF;
   "Tag_5" := "Tag_9" AND NOT #ix_PEC_DiagonallyTT AND NOT #ix_PEC_DetectPackage_1 AND NOT #ix_PEC_DetectPackage_2 AND NOT #ix_PEC_MediumPackage_1;
   IF "Tag_9" AND #ix_PEC_MediumPackage_1 THEN "11-PLC01-CNR06" := 2.0; END_IF;
   "IEC_Counter_0_DB_1".CTU(CU := #ix_PEC_MediumPackage_2, R := #ix_Reset, PV := 10000);
END_REGION

REGION Network 4: big
   IF #sx_Automatic_2 AND "Tag_10" AND (#ix_PEC_DetectPackage_1 OR #ix_PEC_DetectPackage_2) AND NOT #ix_PEC_BigPackage_1 THEN
       #qx_TTForward := TRUE;
       #qx_TTBackward := FALSE;
   END_IF;
   #_w1 := "Tag_10" AND #ix_PEC_BigPackage_1;
   IF #_w1 THEN "11-PLC01-CNR05" := 2.0; END_IF;
   IF #_w1 AND NOT #ix_PEC_DetectPackage_2 THEN
       #qx_TTForward := FALSE;
       #qx_TTBackward := FALSE;
   END_IF;
   "Tag_14" := "Tag_10" AND NOT #ix_PEC_DiagonallyTT AND NOT #ix_PEC_DetectPackage_1 AND NOT #ix_PEC_DetectPackage_2 AND NOT #ix_PEC_DetectPackage_1;
   "IEC_Counter_0_DB_2".CTU(CU := #ix_PEC_BigPackage_2, R := #ix_Reset, PV := 10000);
END_REGION

REGION Network 5
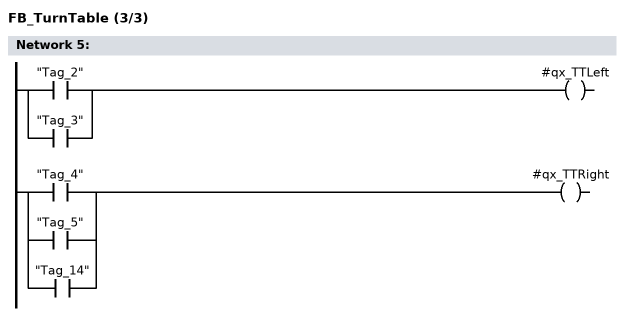
   RUNG wire#powerrail
      Contact( "Tag_2" )
      wire#w1
      Coil( #qx_TTLeft )
   END_RUNG
   RUNG wire#powerrail
      Contact( "Tag_3" )
   END_RUNG wire#w1
   RUNG wire#powerrail
      Contact( "Tag_4" )
      wire#w2
      Coil( #qx_TTRight )
   END_RUNG
   RUNG wire#powerrail
      Contact( "Tag_5" )
   END_RUNG wire#w2
   RUNG wire#powerrail
      Contact( "Tag_14" )
   END_RUNG wire#w2
   // the same network as SCL:
   #qx_TTLeft := "Tag_2" OR "Tag_3";
   #qx_TTRight := "Tag_4" OR "Tag_5" OR "Tag_14";
END_REGION
END_FUNCTION_BLOCK

FUNCTION_BLOCK "FD_FIFO"   // FB6, LAD
{ S7_Optimized_Access := 'TRUE' }
VERSION : 0.1
   VAR
      si_RetVal : Int;
      si_Pointer : Int := 0;
      si_RetVal2 : Int;
      si : Int;
      sx_dupa : Bool;
      sx_dupa2 : Bool;
   END_VAR
   VAR_TEMP   // added for the SCL form of the ladder/FBD networks
      _w1 : Bool;
   END_VAR
BEGIN

REGION Network 1
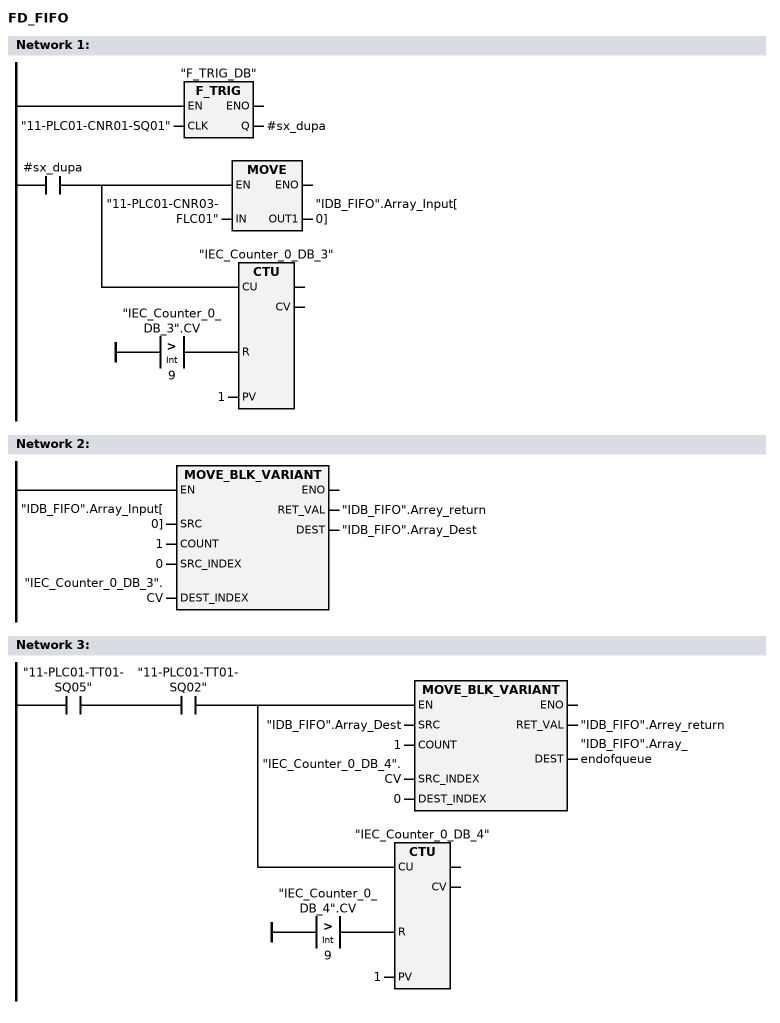
   "F_TRIG_DB"(CLK := "11-PLC01-CNR01-SQ01", Q => #sx_dupa);   // F_TRIG
   IF #sx_dupa THEN "IDB_FIFO".Array_Input[0] := "11-PLC01-CNR03-FLC01"; END_IF;
   "IEC_Counter_0_DB_3".CTU(CU := #sx_dupa, R := "IEC_Counter_0_DB_3".CV > 9, PV := 1);
END_REGION

REGION Network 2
   "IDB_FIFO".Arrey_return := MOVE_BLK_VARIANT(SRC := "IDB_FIFO".Array_Input[0],
                           COUNT := 1,
                           SRC_INDEX := 0,
                           DEST_INDEX := "IEC_Counter_0_DB_3".CV,
                           DEST => "IDB_FIFO".Array_Dest);
END_REGION

REGION Network 3
   #_w1 := "11-PLC01-TT01-SQ05" AND "11-PLC01-TT01-SQ02";
   IF #_w1 THEN
       "IDB_FIFO".Arrey_return := MOVE_BLK_VARIANT(SRC := "IDB_FIFO".Array_Dest,
                               COUNT := 1,
                               SRC_INDEX := "IEC_Counter_0_DB_4".CV,
                               DEST_INDEX := 0,
                               DEST => "IDB_FIFO".Array_endofqueue);
   END_IF;
   "IEC_Counter_0_DB_4".CTU(CU := #_w1, R := "IEC_Counter_0_DB_4".CV > 9, PV := 1);
END_REGION
END_FUNCTION_BLOCK

FUNCTION_BLOCK "FB_Sequence"   // FB7, GRAPH_PLUS
{ S7_Optimized_Access := 'TRUE' }
VERSION : 0.1
   VAR_INPUT
      OFF_SQ : Bool := false;   // Turn sequence off
      INIT_SQ : Bool := false;   // Set sequence to initial state
      ACK_EF : Bool := false;   // Acknowledge all errors and faults
      S_PREV : Bool := false;   // Output previous step in parameter S_NO
      S_NEXT : Bool := false;   // Indicate next step in parameter S_NO
      SW_AUTO : Bool := false;   // Automatic mode
      SW_TAP : Bool := false;   // Semiautomatic/switch with transition
      SW_TOP : Bool := false;   // Semiautomatic/ignore transition
      SW_MAN : Bool := false;   // Manual mode
      S_SEL : Int := 0;   // Select step to be output to S_NO
      S_ON : Bool := false;   // Activate step indicated in S_NO
      S_OFF : Bool := false;   // Deactivate step indicated S_NO
      T_PUSH : Bool := false;   // Enable transition to switch in semi automatic mode
   END_VAR
   VAR_OUTPUT
      S_NO : Int := 0;   // Step number
      S_MORE : Bool := false;   // More steps are available and can be shown in S_NO
      S_ACTIVE : Bool := false;   // Step indicated in S_NO is active
      ERR_FLT : Bool := false;   // Interlock or supervision group error
      AUTO_ON : Bool := false;   // Automatic mode is active
      TAP_ON : Bool := false;   // Semiautomatic mode/step with transition enabled
      TOP_ON : Bool := false;   // Semiautomatic mode/ignore transition enabled
      MAN_ON : Bool := false;   // Manual mode is active
   END_VAR
   VAR
      HMI_INFO : Array[0..11] of UInt;
      IF_PAR : G7_IfParPlus_V6;
      RT_DATA : G7_RTDataPlus_V6;   // Internal data area
      Trans1 : G7_TransitionPlus_V6;   // Transition structure
      Trans2 : G7_TransitionPlus_V6;   // Transition structure
      Trans3 : G7_TransitionPlus_V6;   // Transition structure
      Trans4 : G7_TransitionPlus_V6;   // Transition structure
      Trans5 : G7_TransitionPlus_V6;   // Transition structure
      Trans6 : G7_TransitionPlus_V6;   // Transition structure
      Trans7 : G7_TransitionPlus_V6;   // Transition structure
      Trans8 : G7_TransitionPlus_V6;   // Transition structure
      Trans9 : G7_TransitionPlus_V6;   // Transition structure
      Trans10 : G7_TransitionPlus_V6;   // Transition structure
      Trans11 : G7_TransitionPlus_V6;   // Transition structure
      Trans12 : G7_TransitionPlus_V6;   // Transition structure
      Trans13 : G7_TransitionPlus_V6;   // Transition structure
      Trans14 : G7_TransitionPlus_V6;   // Transition structure
      Trans15 : G7_TransitionPlus_V6;   // Transition structure
      Step1 : G7_StepPlus_V6;   // Step structure
      Step2 : G7_StepPlus_V6;   // Step structure
      Step3 : G7_StepPlus_V6;   // Step structure
      Step4 : G7_StepPlus_V6;   // Step structure
      Step5 : G7_StepPlus_V6;   // Step structure
      Step6 : G7_StepPlus_V6;   // Step structure
      Step7 : G7_StepPlus_V6;   // Step structure
      Step8 : G7_StepPlus_V6;   // Step structure
      Step9 : G7_StepPlus_V6;   // Step structure
      Step10 : G7_StepPlus_V6;   // Step structure
      Step11 : G7_StepPlus_V6;   // Step structure
      Step12 : G7_StepPlus_V6;   // Step structure
      Step13 : G7_StepPlus_V6;   // Step structure
      Step14 : G7_StepPlus_V6;   // Step structure
      Step15 : G7_StepPlus_V6;   // Step structure
      SINI : Array[0..4] of USInt;
      LSTT : Array[0..14] of USInt;
      ATAJ : Array[0..14] of USInt;
      ATAB : Array[0..14] of USInt;
      PSTT : Array[0..14] of USInt;
      NSTT : Array[0..14] of USInt;
      ASSJ : Array[0..14] of USInt;
      ASSB : Array[0..14] of USInt;
      PTTS : Array[0..14] of USInt;
      NTTS : Array[0..14] of USInt;
      SW_SQTS : Array[0..14] of USInt;
      SWITCH : Array[0..1] of USInt;
      TVX : Array[0..4] of USInt;
      TTX : Array[0..4] of USInt;
      TSX : Array[0..4] of USInt;
      S00X : Array[0..4] of USInt;
      SOFFX : Array[0..4] of USInt;
      SONX : Array[0..4] of USInt;
      SAX : Array[0..4] of USInt;
      SERRX : Array[0..15] of USInt;
      SMX : Array[0..15] of USInt;
      S0X : Array[0..15] of USInt;
      S1X : Array[0..15] of USInt;
      IL_ALARM_INST : Diag_Alarm;
      SUP_ALARM_INST : Diag_Alarm;
      STEP_TIME_ALARM_INST : Diag_Alarm;
      IEC_TIMER_INST : IEC_TIMER;
      TRANSACTION_FLAG : Bool := false;
   END_VAR
   // SINI[0] := 2;
   // SINI[2] := 255;
   // SINI[3] := 255;
   // SINI[4] := 255;
   // LSTT[0] := 255;
   // LSTT[1] := 255;
   // LSTT[2] := 255;
   // LSTT[3] := 255;
   // LSTT[4] := 255;
   // LSTT[5] := 255;
   // LSTT[6] := 255;
   // LSTT[8] := 255;
   // LSTT[9] := 255;
   // LSTT[11] := 255;
   // LSTT[12] := 255;
   // LSTT[13] := 255;
   // ATAJ[1] := 1;
   // ATAJ[2] := 2;
   // ATAJ[3] := 3;
   // ATAJ[4] := 4;
   // ATAJ[5] := 5;
   // ATAJ[6] := 6;
   // ATAJ[7] := 7;
   // ATAJ[8] := 8;
   // ATAJ[9] := 9;
   // ATAJ[10] := 10;
   // ATAJ[11] := 11;
   // ATAJ[12] := 12;
   // ATAJ[13] := 13;
   // ATAJ[14] := 14;
   // ATAB[1] := 1;
   // ATAB[2] := 2;
   // ATAB[3] := 3;
   // ATAB[4] := 4;
   // ATAB[5] := 5;
   // ATAB[6] := 6;
   // ATAB[7] := 7;
   // ATAB[8] := 8;
   // ATAB[9] := 9;
   // ATAB[10] := 10;
   // ATAB[11] := 11;
   // ATAB[12] := 12;
   // ATAB[13] := 13;
   // ATAB[14] := 14;
   // PSTT[1] := 1;
   // PSTT[2] := 2;
   // PSTT[3] := 3;
   // PSTT[4] := 4;
   // PSTT[5] := 5;
   // PSTT[6] := 6;
   // PSTT[7] := 7;
   // PSTT[8] := 8;
   // PSTT[9] := 9;
   // PSTT[10] := 10;
   // PSTT[11] := 11;
   // PSTT[12] := 12;
   // PSTT[13] := 13;
   // PSTT[14] := 14;
   // NSTT[0] := 1;
   // NSTT[1] := 2;
   // NSTT[2] := 3;
   // NSTT[3] := 4;
   // NSTT[4] := 5;
   // NSTT[5] := 6;
   // NSTT[6] := 7;
   // NSTT[8] := 9;
   // NSTT[9] := 10;
   // NSTT[11] := 12;
   // NSTT[12] := 13;
   // NSTT[13] := 14;
   // ASSJ[1] := 1;
   // ASSJ[2] := 2;
   // ASSJ[3] := 3;
   // ASSJ[4] := 4;
   // ASSJ[5] := 5;
   // ASSJ[6] := 6;
   // ASSJ[7] := 7;
   // ASSJ[8] := 8;
   // ASSJ[9] := 9;
   // ASSJ[10] := 10;
   // ASSJ[11] := 11;
   // ASSJ[12] := 12;
   // ASSJ[13] := 13;
   // ASSJ[14] := 14;
   // ASSB[1] := 1;
   // ASSB[2] := 2;
   // ASSB[3] := 3;
   // ASSB[4] := 8;
   // ASSB[5] := 5;
   // ASSB[6] := 6;
   // ASSB[7] := 7;
   // ASSB[8] := 11;
   // ASSB[9] := 9;
   // ASSB[10] := 10;
   // ASSB[11] := 4;
   // ASSB[12] := 12;
   // ASSB[13] := 13;
   // ASSB[14] := 14;
   // PTTS[0] := 255;
   // PTTS[2] := 1;
   // PTTS[3] := 2;
   // PTTS[4] := 3;
   // PTTS[5] := 4;
   // PTTS[6] := 5;
   // PTTS[7] := 6;
   // PTTS[8] := 3;
   // PTTS[9] := 8;
   // PTTS[10] := 9;
   // PTTS[11] := 3;
   // PTTS[12] := 11;
   // PTTS[13] := 12;
   // PTTS[14] := 13;
   // NTTS[1] := 1;
   // NTTS[2] := 2;
   // NTTS[3] := 3;
   // NTTS[4] := 4;
   // NTTS[5] := 5;
   // NTTS[6] := 6;
   // NTTS[7] := 7;
   // NTTS[8] := 8;
   // NTTS[9] := 9;
   // NTTS[10] := 10;
   // NTTS[11] := 11;
   // NTTS[12] := 12;
   // NTTS[13] := 13;
   // NTTS[14] := 14;
   // SW_SQTS[4] := 1;
   // SW_SQTS[5] := 1;
   // SW_SQTS[6] := 1;
   // SW_SQTS[7] := 1;
   // SW_SQTS[8] := 2;
   // SW_SQTS[9] := 2;
   // SW_SQTS[10] := 2;
   // SW_SQTS[11] := 3;
   // SW_SQTS[12] := 3;
   // SW_SQTS[13] := 3;
   // SW_SQTS[14] := 3;
   // SWITCH[0] := 192;
   // SWITCH[1] := 106;
   // TVX[0] := 16#1;
   // TTX[0] := 16#1;
   // TSX[0] := 16#1;
   // S00X[0] := 16#1;
   // SOFFX[0] := 16#1;
   // SONX[0] := 16#1;
   // SAX[0] := 16#1;
   // SERRX[0] := 16#1;
   // SMX[0] := 16#1;
   // S0X[0] := 16#1;
   // S1X[0] := 16#1;
BEGIN
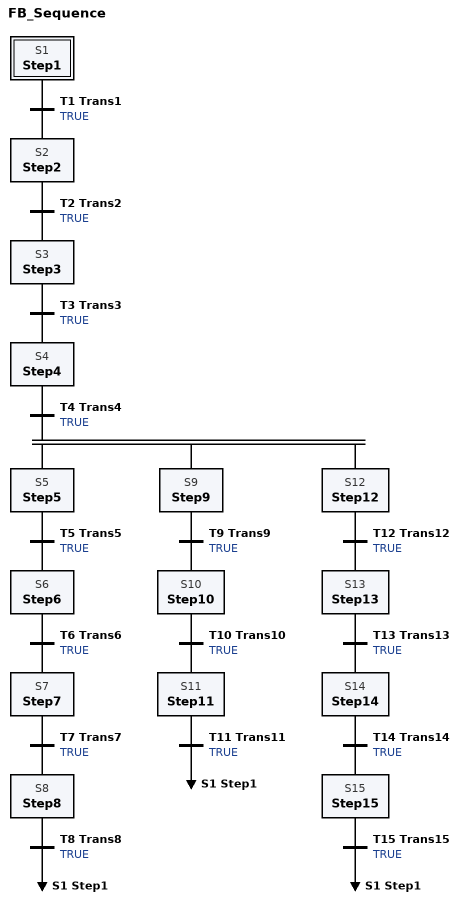
   // sequencer 1
   INITIAL_STEP Step1:   // S1, max time T#10S, warning time T#7S
   END_STEP
   TRANSITION Trans1 FROM Step1 TO Step2   // T1
      := TRUE;
   END_TRANSITION
   STEP Step2:   // S2, max time T#10S, warning time T#7S
   END_STEP
   TRANSITION Trans2 FROM Step2 TO Step3   // T2
      := TRUE;
   END_TRANSITION
   STEP Step3:   // S3, max time T#10S, warning time T#7S
   END_STEP
   TRANSITION Trans3 FROM Step3 TO Step4   // T3
      := TRUE;
   END_TRANSITION
   STEP Step4:   // S4, max time T#10S, warning time T#7S
   END_STEP
   TRANSITION Trans4 FROM Step4 TO (Step5, Step9, Step12)   // T4
      := TRUE;
   END_TRANSITION
   STEP Step5:   // S5, max time T#10S, warning time T#7S
   END_STEP
   TRANSITION Trans5 FROM Step5 TO Step6   // T5
      := TRUE;
   END_TRANSITION
   STEP Step6:   // S6, max time T#10S, warning time T#7S
   END_STEP
   TRANSITION Trans6 FROM Step6 TO Step7   // T6
      := TRUE;
   END_TRANSITION
   STEP Step7:   // S7, max time T#10S, warning time T#7S
   END_STEP
   TRANSITION Trans7 FROM Step7 TO Step8   // T7
      := TRUE;
   END_TRANSITION
   STEP Step8:   // S8, max time T#10S, warning time T#7S
   END_STEP
   TRANSITION Trans8 FROM Step8 TO Step1   // T8, jump
      := TRUE;
   END_TRANSITION
   STEP Step9:   // S9, max time T#10S, warning time T#7S
   END_STEP
   TRANSITION Trans9 FROM Step9 TO Step10   // T9
      := TRUE;
   END_TRANSITION
   STEP Step10:   // S10, max time T#10S, warning time T#7S
   END_STEP
   TRANSITION Trans10 FROM Step10 TO Step11   // T10
      := TRUE;
   END_TRANSITION
   STEP Step11:   // S11, max time T#10S, warning time T#7S
   END_STEP
   TRANSITION Trans11 FROM Step11 TO Step1   // T11, jump
      := TRUE;
   END_TRANSITION
   STEP Step12:   // S12, max time T#10S, warning time T#7S
   END_STEP
   TRANSITION Trans12 FROM Step12 TO Step13   // T12
      := TRUE;
   END_TRANSITION
   STEP Step13:   // S13, max time T#10S, warning time T#7S
   END_STEP
   TRANSITION Trans13 FROM Step13 TO Step14   // T13
      := TRUE;
   END_TRANSITION
   STEP Step14:   // S14, max time T#10S, warning time T#7S
   END_STEP
   TRANSITION Trans14 FROM Step14 TO Step15   // T14
      := TRUE;
   END_TRANSITION
   STEP Step15:   // S15, max time T#10S, warning time T#7S
   END_STEP
   TRANSITION Trans15 FROM Step15 TO Step1   // T15, jump
      := TRUE;
   END_TRANSITION
END_FUNCTION_BLOCK

FUNCTION_BLOCK "FB_Chute"   // FB8, LAD
{ S7_Optimized_Access := 'TRUE' }
VERSION : 0.1
   VAR_INPUT
      ix_Reset_1 : Bool;
      ix_PEC_SmallPackage_2 : Bool;
      ix_PEC_MediumPackage_2 : Bool;
      ix_PEC_BigPackage_2 : Bool;
   END_VAR
   VAR_OUTPUT
      "Small Package" : Int;
      "Medium Package" : Int;
      "Big Package" : Int;
   END_VAR
BEGIN

REGION Network 1
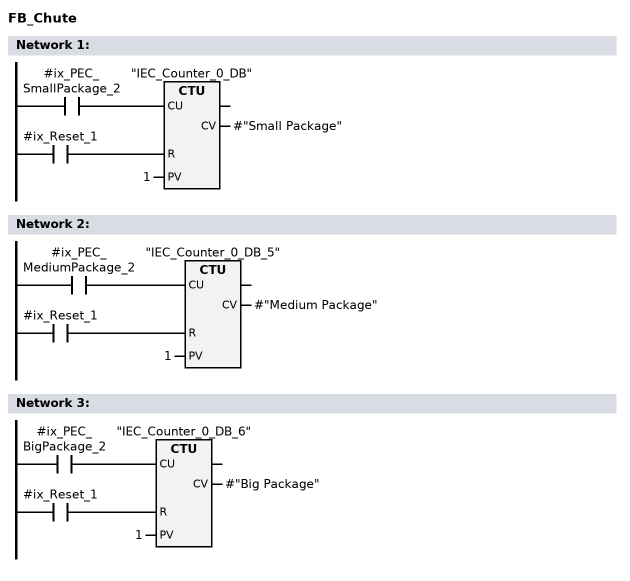
   "IEC_Counter_0_DB".CTU(CU := #ix_PEC_SmallPackage_2, R := #ix_Reset_1, PV := 1, CV => #"Small Package");
END_REGION

REGION Network 2
   "IEC_Counter_0_DB_5".CTU(CU := #ix_PEC_MediumPackage_2, R := #ix_Reset_1, PV := 1, CV => #"Medium Package");
END_REGION

REGION Network 3
   "IEC_Counter_0_DB_6".CTU(CU := #ix_PEC_BigPackage_2, R := #ix_Reset_1, PV := 1, CV => #"Big Package");
END_REGION
END_FUNCTION_BLOCK

FUNCTION "FC_Area" : Void   // FC1, LAD
{ S7_Optimized_Access := 'TRUE' }
VERSION : 0.1
BEGIN

REGION Network 1
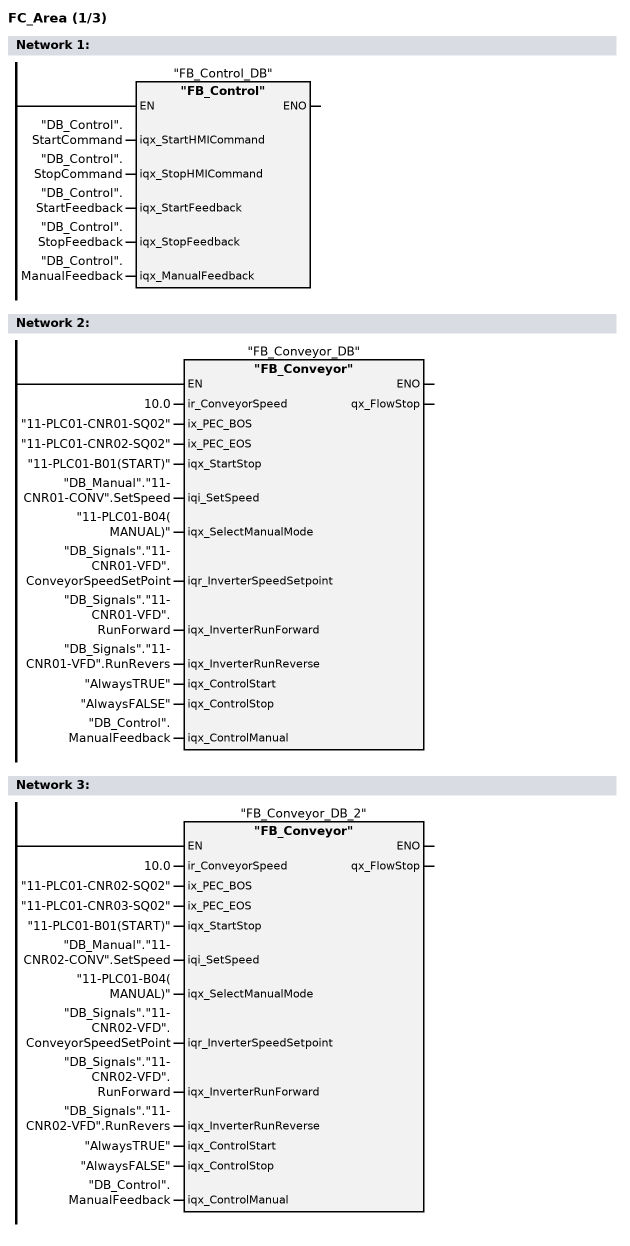
   RUNG wire#powerrail
      "FB_Control_DB"(iqx_StartHMICommand := "DB_Control".StartCommand, iqx_StopHMICommand := "DB_Control".StopCommand, iqx_StartFeedback := "DB_Control".StartFeedback, iqx_StopFeedback := "DB_Control".StopFeedback, iqx_ManualFeedback := "DB_Control".ManualFeedback)
   END_RUNG
   // the same network as SCL:
   "FB_Control_DB"(iqx_StartHMICommand := "DB_Control".StartCommand,   // "FB_Control"
                   iqx_StopHMICommand := "DB_Control".StopCommand,
                   iqx_StartFeedback := "DB_Control".StartFeedback,
                   iqx_StopFeedback := "DB_Control".StopFeedback,
                   iqx_ManualFeedback := "DB_Control".ManualFeedback);
END_REGION

REGION Network 2
   RUNG wire#powerrail
      "FB_Conveyor_DB"(ir_ConveyorSpeed := 10.0, ix_PEC_BOS := "11-PLC01-CNR01-SQ02", ix_PEC_EOS := "11-PLC01-CNR02-SQ02", iqx_StartStop := "11-PLC01-B01(START)", iqi_SetSpeed := "DB_Manual"."11-CNR01-CONV".SetSpeed, iqx_SelectManualMode := "11-PLC01-B04(MANUAL)", iqr_InverterSpeedSetpoint := "DB_Signals"."11-CNR01-VFD".ConveyorSpeedSetPoint, iqx_InverterRunForward := "DB_Signals"."11-CNR01-VFD".RunForward, iqx_InverterRunReverse := "DB_Signals"."11-CNR01-VFD".RunRevers, iqx_ControlStart := "AlwaysTRUE", iqx_ControlStop := "AlwaysFALSE", iqx_ControlManual := "DB_Control".ManualFeedback, qx_FlowStop =>)
   END_RUNG
   // the same network as SCL:
   "FB_Conveyor_DB"(ir_ConveyorSpeed := 10.0,   // "FB_Conveyor"
                    ix_PEC_BOS := "11-PLC01-CNR01-SQ02",
                    ix_PEC_EOS := "11-PLC01-CNR02-SQ02",
                    iqx_StartStop := "11-PLC01-B01(START)",
                    iqi_SetSpeed := "DB_Manual"."11-CNR01-CONV".SetSpeed,
                    iqx_SelectManualMode := "11-PLC01-B04(MANUAL)",
                    iqr_InverterSpeedSetpoint := "DB_Signals"."11-CNR01-VFD".ConveyorSpeedSetPoint,
                    iqx_InverterRunForward := "DB_Signals"."11-CNR01-VFD".RunForward,
                    iqx_InverterRunReverse := "DB_Signals"."11-CNR01-VFD".RunRevers,
                    iqx_ControlStart := "AlwaysTRUE",
                    iqx_ControlStop := "AlwaysFALSE",
                    iqx_ControlManual := "DB_Control".ManualFeedback);
END_REGION

REGION Network 3
   RUNG wire#powerrail
      "FB_Conveyor_DB_2"(ir_ConveyorSpeed := 10.0, ix_PEC_BOS := "11-PLC01-CNR02-SQ02", ix_PEC_EOS := "11-PLC01-CNR03-SQ02", iqx_StartStop := "11-PLC01-B01(START)", iqi_SetSpeed := "DB_Manual"."11-CNR02-CONV".SetSpeed, iqx_SelectManualMode := "11-PLC01-B04(MANUAL)", iqr_InverterSpeedSetpoint := "DB_Signals"."11-CNR02-VFD".ConveyorSpeedSetPoint, iqx_InverterRunForward := "DB_Signals"."11-CNR02-VFD".RunForward, iqx_InverterRunReverse := "DB_Signals"."11-CNR02-VFD".RunRevers, iqx_ControlStart := "AlwaysTRUE", iqx_ControlStop := "AlwaysFALSE", iqx_ControlManual := "DB_Control".ManualFeedback, qx_FlowStop =>)
   END_RUNG
   // the same network as SCL:
   "FB_Conveyor_DB_2"(ir_ConveyorSpeed := 10.0,   // "FB_Conveyor"
                      ix_PEC_BOS := "11-PLC01-CNR02-SQ02",
                      ix_PEC_EOS := "11-PLC01-CNR03-SQ02",
                      iqx_StartStop := "11-PLC01-B01(START)",
                      iqi_SetSpeed := "DB_Manual"."11-CNR02-CONV".SetSpeed,
                      iqx_SelectManualMode := "11-PLC01-B04(MANUAL)",
                      iqr_InverterSpeedSetpoint := "DB_Signals"."11-CNR02-VFD".ConveyorSpeedSetPoint,
                      iqx_InverterRunForward := "DB_Signals"."11-CNR02-VFD".RunForward,
                      iqx_InverterRunReverse := "DB_Signals"."11-CNR02-VFD".RunRevers,
                      iqx_ControlStart := "AlwaysTRUE",
                      iqx_ControlStop := "AlwaysFALSE",
                      iqx_ControlManual := "DB_Control".ManualFeedback);
END_REGION

REGION Network 4
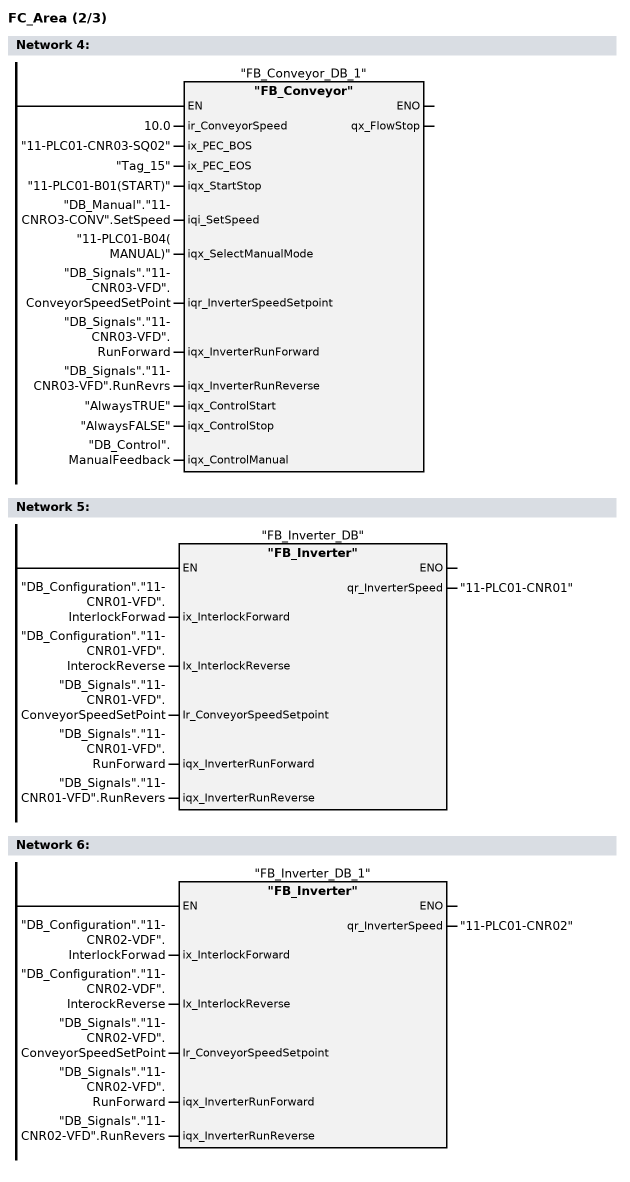
   RUNG wire#powerrail
      "FB_Conveyor_DB_1"(ir_ConveyorSpeed := 10.0, ix_PEC_BOS := "11-PLC01-CNR03-SQ02", ix_PEC_EOS := "Tag_15", iqx_StartStop := "11-PLC01-B01(START)", iqi_SetSpeed := "DB_Manual"."11-CNRO3-CONV".SetSpeed, iqx_SelectManualMode := "11-PLC01-B04(MANUAL)", iqr_InverterSpeedSetpoint := "DB_Signals"."11-CNR03-VFD".ConveyorSpeedSetPoint, iqx_InverterRunForward := "DB_Signals"."11-CNR03-VFD".RunForward, iqx_InverterRunReverse := "DB_Signals"."11-CNR03-VFD".RunRevrs, iqx_ControlStart := "AlwaysTRUE", iqx_ControlStop := "AlwaysFALSE", iqx_ControlManual := "DB_Control".ManualFeedback, qx_FlowStop =>)
   END_RUNG
   // the same network as SCL:
   "FB_Conveyor_DB_1"(ir_ConveyorSpeed := 10.0,   // "FB_Conveyor"
                      ix_PEC_BOS := "11-PLC01-CNR03-SQ02",
                      ix_PEC_EOS := "Tag_15",
                      iqx_StartStop := "11-PLC01-B01(START)",
                      iqi_SetSpeed := "DB_Manual"."11-CNRO3-CONV".SetSpeed,
                      iqx_SelectManualMode := "11-PLC01-B04(MANUAL)",
                      iqr_InverterSpeedSetpoint := "DB_Signals"."11-CNR03-VFD".ConveyorSpeedSetPoint,
                      iqx_InverterRunForward := "DB_Signals"."11-CNR03-VFD".RunForward,
                      iqx_InverterRunReverse := "DB_Signals"."11-CNR03-VFD".RunRevrs,
                      iqx_ControlStart := "AlwaysTRUE",
                      iqx_ControlStop := "AlwaysFALSE",
                      iqx_ControlManual := "DB_Control".ManualFeedback);
END_REGION

REGION Network 5
   RUNG wire#powerrail
      "FB_Inverter_DB"(ix_InterlockForward := "DB_Configuration"."11-CNR01-VFD".InterlockForwad, Ix_InterlockReverse := "DB_Configuration"."11-CNR01-VFD".InterockReverse, Ir_ConveyorSpeedSetpoint := "DB_Signals"."11-CNR01-VFD".ConveyorSpeedSetPoint, iqx_InverterRunForward := "DB_Signals"."11-CNR01-VFD".RunForward, iqx_InverterRunReverse := "DB_Signals"."11-CNR01-VFD".RunRevers, qr_InverterSpeed => "11-PLC01-CNR01")
   END_RUNG
   // the same network as SCL:
   "FB_Inverter_DB"(ix_InterlockForward := "DB_Configuration"."11-CNR01-VFD".InterlockForwad,   // "FB_Inverter"
                    Ix_InterlockReverse := "DB_Configuration"."11-CNR01-VFD".InterockReverse,
                    Ir_ConveyorSpeedSetpoint := "DB_Signals"."11-CNR01-VFD".ConveyorSpeedSetPoint,
                    iqx_InverterRunForward := "DB_Signals"."11-CNR01-VFD".RunForward,
                    iqx_InverterRunReverse := "DB_Signals"."11-CNR01-VFD".RunRevers,
                    qr_InverterSpeed => "11-PLC01-CNR01");
END_REGION

REGION Network 6
   RUNG wire#powerrail
      "FB_Inverter_DB_1"(ix_InterlockForward := "DB_Configuration"."11-CNR02-VDF".InterlockForwad, Ix_InterlockReverse := "DB_Configuration"."11-CNR02-VDF".InterockReverse, Ir_ConveyorSpeedSetpoint := "DB_Signals"."11-CNR02-VFD".ConveyorSpeedSetPoint, iqx_InverterRunForward := "DB_Signals"."11-CNR02-VFD".RunForward, iqx_InverterRunReverse := "DB_Signals"."11-CNR02-VFD".RunRevers, qr_InverterSpeed => "11-PLC01-CNR02")
   END_RUNG
   // the same network as SCL:
   "FB_Inverter_DB_1"(ix_InterlockForward := "DB_Configuration"."11-CNR02-VDF".InterlockForwad,   // "FB_Inverter"
                      Ix_InterlockReverse := "DB_Configuration"."11-CNR02-VDF".InterockReverse,
                      Ir_ConveyorSpeedSetpoint := "DB_Signals"."11-CNR02-VFD".ConveyorSpeedSetPoint,
                      iqx_InverterRunForward := "DB_Signals"."11-CNR02-VFD".RunForward,
                      iqx_InverterRunReverse := "DB_Signals"."11-CNR02-VFD".RunRevers,
                      qr_InverterSpeed => "11-PLC01-CNR02");
END_REGION

REGION Network 7
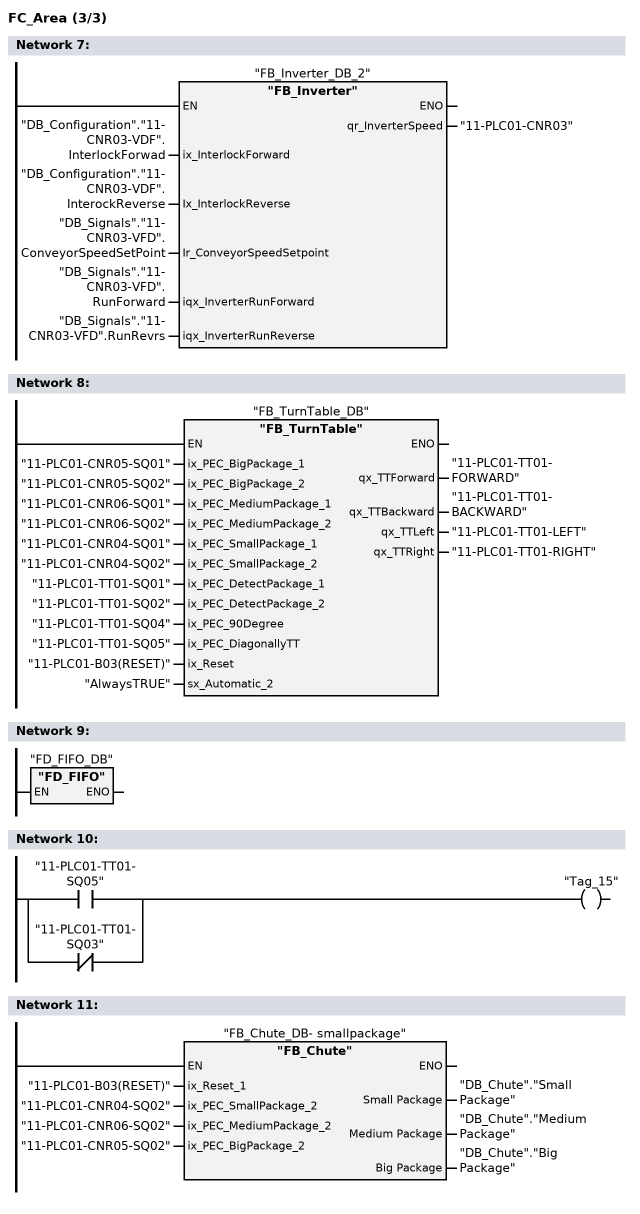
   RUNG wire#powerrail
      "FB_Inverter_DB_2"(ix_InterlockForward := "DB_Configuration"."11-CNR03-VDF".InterlockForwad, Ix_InterlockReverse := "DB_Configuration"."11-CNR03-VDF".InterockReverse, Ir_ConveyorSpeedSetpoint := "DB_Signals"."11-CNR03-VFD".ConveyorSpeedSetPoint, iqx_InverterRunForward := "DB_Signals"."11-CNR03-VFD".RunForward, iqx_InverterRunReverse := "DB_Signals"."11-CNR03-VFD".RunRevrs, qr_InverterSpeed => "11-PLC01-CNR03")
   END_RUNG
   // the same network as SCL:
   "FB_Inverter_DB_2"(ix_InterlockForward := "DB_Configuration"."11-CNR03-VDF".InterlockForwad,   // "FB_Inverter"
                      Ix_InterlockReverse := "DB_Configuration"."11-CNR03-VDF".InterockReverse,
                      Ir_ConveyorSpeedSetpoint := "DB_Signals"."11-CNR03-VFD".ConveyorSpeedSetPoint,
                      iqx_InverterRunForward := "DB_Signals"."11-CNR03-VFD".RunForward,
                      iqx_InverterRunReverse := "DB_Signals"."11-CNR03-VFD".RunRevrs,
                      qr_InverterSpeed => "11-PLC01-CNR03");
END_REGION

REGION Network 8
   RUNG wire#powerrail
      "FB_TurnTable_DB"(ix_PEC_BigPackage_1 := "11-PLC01-CNR05-SQ01", ix_PEC_BigPackage_2 := "11-PLC01-CNR05-SQ02", ix_PEC_MediumPackage_1 := "11-PLC01-CNR06-SQ01", ix_PEC_MediumPackage_2 := "11-PLC01-CNR06-SQ02", ix_PEC_SmallPackage_1 := "11-PLC01-CNR04-SQ01", ix_PEC_SmallPackage_2 := "11-PLC01-CNR04-SQ02", ix_PEC_DetectPackage_1 := "11-PLC01-TT01-SQ01", ix_PEC_DetectPackage_2 := "11-PLC01-TT01-SQ02", ix_PEC_90Degree := "11-PLC01-TT01-SQ04", ix_PEC_DiagonallyTT := "11-PLC01-TT01-SQ05", ix_Reset := "11-PLC01-B03(RESET)", sx_Automatic_2 := "AlwaysTRUE", qx_TTForward => "11-PLC01-TT01-FORWARD", qx_TTBackward => "11-PLC01-TT01-BACKWARD", qx_TTLeft => "11-PLC01-TT01-LEFT", qx_TTRight => "11-PLC01-TT01-RIGHT")
   END_RUNG
   // the same network as SCL:
   "FB_TurnTable_DB"(ix_PEC_BigPackage_1 := "11-PLC01-CNR05-SQ01",   // "FB_TurnTable"
                     ix_PEC_BigPackage_2 := "11-PLC01-CNR05-SQ02",
                     ix_PEC_MediumPackage_1 := "11-PLC01-CNR06-SQ01",
                     ix_PEC_MediumPackage_2 := "11-PLC01-CNR06-SQ02",
                     ix_PEC_SmallPackage_1 := "11-PLC01-CNR04-SQ01",
                     ix_PEC_SmallPackage_2 := "11-PLC01-CNR04-SQ02",
                     ix_PEC_DetectPackage_1 := "11-PLC01-TT01-SQ01",
                     ix_PEC_DetectPackage_2 := "11-PLC01-TT01-SQ02",
                     ix_PEC_90Degree := "11-PLC01-TT01-SQ04",
                     ix_PEC_DiagonallyTT := "11-PLC01-TT01-SQ05",
                     ix_Reset := "11-PLC01-B03(RESET)",
                     sx_Automatic_2 := "AlwaysTRUE",
                     qx_TTForward => "11-PLC01-TT01-FORWARD",
                     qx_TTBackward => "11-PLC01-TT01-BACKWARD",
                     qx_TTLeft => "11-PLC01-TT01-LEFT",
                     qx_TTRight => "11-PLC01-TT01-RIGHT");
END_REGION

REGION Network 9
   RUNG wire#powerrail
      "FD_FIFO_DB"()
   END_RUNG
   // the same network as SCL:
   "FD_FIFO_DB"();   // "FD_FIFO"
END_REGION

REGION Network 10
   RUNG wire#powerrail
      Contact( "11-PLC01-TT01-SQ05" )
      wire#w1
      Coil( "Tag_15" )
   END_RUNG
   RUNG wire#powerrail
      I_Contact( "11-PLC01-TT01-SQ03" )
   END_RUNG wire#w1
   // the same network as SCL:
   "Tag_15" := "11-PLC01-TT01-SQ05" OR NOT "11-PLC01-TT01-SQ03";
END_REGION

REGION Network 11
   RUNG wire#powerrail
      "FB_Chute_DB- smallpackage"(ix_Reset_1 := "11-PLC01-B03(RESET)", ix_PEC_SmallPackage_2 := "11-PLC01-CNR04-SQ02", ix_PEC_MediumPackage_2 := "11-PLC01-CNR06-SQ02", ix_PEC_BigPackage_2 := "11-PLC01-CNR05-SQ02", "Small Package" => "DB_Chute"."Small Package", "Medium Package" => "DB_Chute"."Medium Package", "Big Package" => "DB_Chute"."Big Package")
   END_RUNG
   // the same network as SCL:
   "FB_Chute_DB- smallpackage"(ix_Reset_1 := "11-PLC01-B03(RESET)",   // "FB_Chute"
                           ix_PEC_SmallPackage_2 := "11-PLC01-CNR04-SQ02",
                           ix_PEC_MediumPackage_2 := "11-PLC01-CNR06-SQ02",
                           ix_PEC_BigPackage_2 := "11-PLC01-CNR05-SQ02",
                           "Small Package" => "DB_Chute"."Small Package",
                           "Medium Package" => "DB_Chute"."Medium Package",
                           "Big Package" => "DB_Chute"."Big Package");
END_REGION
END_FUNCTION

ORGANIZATION_BLOCK "Main"   // OB1, LAD, ProgramCycle
TITLE = "Main Program Sweep (Cycle)"
{ S7_Optimized_Access := 'TRUE' }
VERSION : 0.1
   VAR_INPUT
      Initial_Call : Bool;   // Initial call of this OB
      Remanence : Bool;   // =True, if remanent data are available
   END_VAR
BEGIN

REGION Network 1
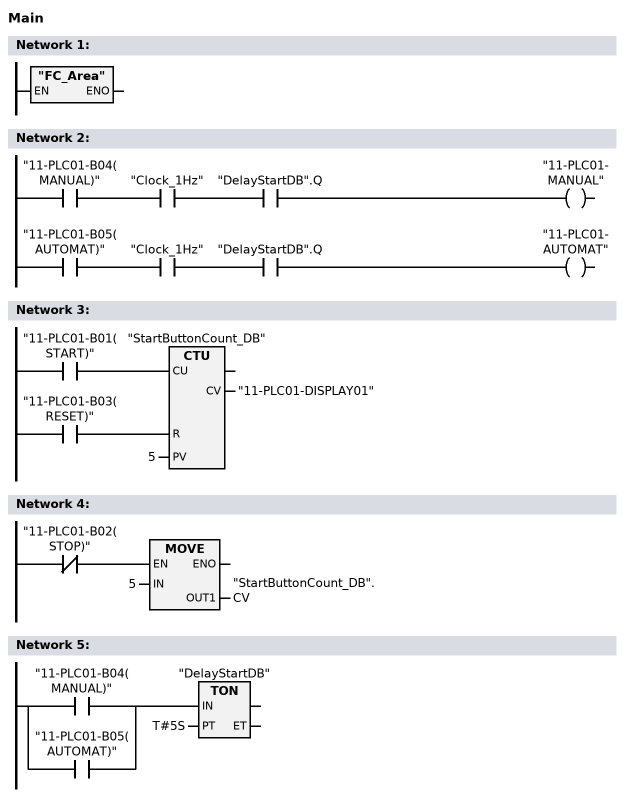
   RUNG wire#powerrail
      "FC_Area"()
   END_RUNG
   // the same network as SCL:
   "FC_Area"();
END_REGION

REGION Network 2
   RUNG wire#powerrail
      Contact( "11-PLC01-B04(MANUAL)" )
      Contact( "Clock_1Hz" )
      Contact( "DelayStartDB".Q )
      Coil( "11-PLC01-MANUAL" )
   END_RUNG
   RUNG wire#powerrail
      Contact( "11-PLC01-B05(AUTOMAT)" )
      Contact( "Clock_1Hz" )
      Contact( "DelayStartDB".Q )
      Coil( "11-PLC01-AUTOMAT" )
   END_RUNG
   // the same network as SCL:
   "11-PLC01-MANUAL" := "11-PLC01-B04(MANUAL)" AND "Clock_1Hz" AND "DelayStartDB".Q;
   "11-PLC01-AUTOMAT" := "11-PLC01-B05(AUTOMAT)" AND "Clock_1Hz" AND "DelayStartDB".Q;
END_REGION

REGION Network 3
   "StartButtonCount_DB".CTU(CU := "11-PLC01-B01(START)",
                           R := "11-PLC01-B03(RESET)",
                           PV := 5,
                           CV => "11-PLC01-DISPLAY01");
END_REGION

REGION Network 4
   RUNG wire#powerrail
      I_Contact( "11-PLC01-B02(STOP)" )
      Move(in := 5, out1 => "StartButtonCount_DB".CV)
   END_RUNG
   // the same network as SCL:
   IF NOT "11-PLC01-B02(STOP)" THEN "StartButtonCount_DB".CV := 5; END_IF;
END_REGION

REGION Network 5
   "DelayStartDB".TON(IN := "11-PLC01-B04(MANUAL)" OR "11-PLC01-B05(AUTOMAT)", PT := T#5S);
END_REGION
END_ORGANIZATION_BLOCK